// NodeFactory/Datatype/DatatypeNodeFactory
{attribute 'linkalways'} 
{attribute 'no_explicit_call' := 'This FB is a CLASS and must be accessed using methods or properties'}
{attribute 'enable_dynamic_creation'}
FUNCTION_BLOCK DatatypeNodeFactory IMPLEMENTS I_EventHandler
VAR
	datatypes : I_Datatypes;
	nodeFactory : I_NodeFactory;
	selfCreatedNodes : Stack;
END_VAR

METHOD FB_init : BOOL
VAR_INPUT
	bInitRetains : BOOL; // if TRUE, the retain variables are initialized (warm start / cold start)
	bInCopyCode : BOOL;  // if TRUE, the instance afterwards gets moved into the copy code (online change)
	Datatypes : I_Datatypes;
	NodeFactory : I_NodeFactory;	
END_VAR
THIS^.datatypes := Datatypes;
THIS^.nodeFactory := NodeFactory;

RegisterWithDatatypes();
END_METHOD

METHOD FB_exit : BOOL
VAR_INPUT
	bInCopyCode : BOOL; // if TRUE, the exit method is called for exiting an instance that is copied afterwards (online change).
END_VAR
IF bInCopyCode THEN
	RETURN;
END_IF

DeregisterWithDatatypes();
DisposeSelfCreatedNodes();
END_METHOD

METHOD PRIVATE DeregisterWithDatatypes
VAR_INPUT
END_VAR
IF datatypes = 0 THEN
	RETURN;
END_IF

datatypes.OffEvent('OnDatatypeAdded', THIS^);
datatypes := 0;
END_METHOD

METHOD PRIVATE DisposeSelfCreatedNodes : BOOL
VAR
	node : I_Node;
END_VAR
WHILE selfCreatedNodes.TryPop(node) DO
	node.Dispose();
END_WHILE
END_METHOD

METHOD PRIVATE RegisterWithDatatypes
VAR_INPUT
END_VAR
IF datatypes = 0 THEN
	RETURN;
END_IF

datatypes.OnEvent('OnDatatypeAdded', THIS^);
END_METHOD

METHOD PROTECTED CreateAliasArrayBundleNode : I_Node
VAR_INPUT
	NodeDatatype : I_AliasDatatype;
END_VAR
VAR
	pAnyBundleNode : POINTER TO AnyAliasArrayBundleNode;
END_VAR
pAnyBundleNode := __NEW(AnyAliasArrayBundleNode(AliasDatatype := NodeDatatype));
CreateAliasArrayBundleNode := pAnyBundleNode^;
END_METHOD

METHOD PROTECTED CreateAliasArrayUnbundleNode : I_Node
VAR_INPUT
	NodeDatatype : I_AliasDatatype;
END_VAR
VAR
	pAnyUnbundleNode : POINTER TO AnyAliasArrayUnbundleNode;
END_VAR
pAnyUnbundleNode := __NEW(AnyAliasArrayUnbundleNode(AliasDatatype := NodeDatatype));
CreateAliasArrayUnbundleNode := pAnyUnbundleNode^;
END_METHOD

METHOD PROTECTED CreateAliasStructureBundleNode : I_Node
VAR_INPUT
	NodeDatatype : I_AliasDatatype;
END_VAR
VAR
	pAnyBundleNode : POINTER TO AnyAliasStructureBundleNode;
END_VAR
pAnyBundleNode := __NEW(AnyAliasStructureBundleNode(AliasDatatype := NodeDatatype));
CreateAliasStructureBundleNode := pAnyBundleNode^;
END_METHOD

METHOD PROTECTED CreateAliasStructureUnbundleNode : I_Node
VAR_INPUT
	NodeDatatype : I_AliasDatatype;
END_VAR
VAR
	pAnyUnbundleNode : POINTER TO AnyAliasStructureUnbundleNode;
END_VAR
pAnyUnbundleNode := __NEW(AnyAliasStructureUnbundleNode(AliasDatatype := NodeDatatype));
CreateAliasStructureUnbundleNode := pAnyUnbundleNode^;
END_METHOD

METHOD PROTECTED CreateArrayBundleNode : I_Node
VAR_INPUT
	NodeDatatype : I_ArrayDatatype;
END_VAR
VAR
	pAnyBundleNode : POINTER TO AnyArrayBundleNode;
END_VAR
pAnyBundleNode := __NEW(AnyArrayBundleNode(ArrayDatatype := NodeDatatype));
CreateArrayBundleNode := pAnyBundleNode^;
END_METHOD

METHOD PROTECTED CreateArrayUnbundleNode : I_Node
VAR_INPUT
	NodeDatatype : I_ArrayDatatype;
END_VAR
VAR
	pAnyUnbundleNode : POINTER TO AnyArrayUnbundleNode;
END_VAR
pAnyUnbundleNode := __NEW(AnyArrayUnbundleNode(ArrayDatatype := NodeDatatype));
CreateArrayUnbundleNode := pAnyUnbundleNode^;
END_METHOD

METHOD PROTECTED CreateDisplayNode : I_Node
VAR_INPUT
	NodeDatatype : I_Datatype;
END_VAR
VAR
	pAnyDisplayNode : POINTER TO AnyDisplayNode;
END_VAR
pAnyDisplayNode := __NEW(AnyDisplayNode(Datatype := NodeDatatype));
CreateDisplayNode := pAnyDisplayNode^;
END_METHOD

METHOD PROTECTED CreateInterfaceDisplayNode : I_Node
VAR_INPUT
	NodeDatatype : I_InterfaceDatatype;
END_VAR
VAR
	pAnyInterfaceDisplayNode : POINTER TO AnyInterfaceDisplayNode;
END_VAR
pAnyInterfaceDisplayNode := __NEW(AnyInterfaceDisplayNode(Datatype := NodeDatatype));
CreateInterfaceDisplayNode := pAnyInterfaceDisplayNode^;
END_METHOD

METHOD PROTECTED CreateLiteralNode : I_Node
VAR_INPUT
	NodeDatatype : I_Datatype;
END_VAR
VAR
	pAnyLiteralNode : POINTER TO AnyLiteralNode;
END_VAR
pAnyLiteralNode := __NEW(AnyLiteralNode(Datatype := NodeDatatype));
CreateLiteralNode := pAnyLiteralNode^;
END_METHOD

METHOD PROTECTED CreateStructureBundleNode : I_Node
VAR_INPUT
	NodeDatatype : I_StructuredDatatype;
END_VAR
VAR
	pAnyBundleNode : POINTER TO AnyStructureBundleNode;
END_VAR
pAnyBundleNode := __NEW(AnyStructureBundleNode(StructuredDatatype := NodeDatatype));
CreateStructureBundleNode := pAnyBundleNode^;
END_METHOD

METHOD PROTECTED CreateStructureUnbundleNode : I_Node
VAR_INPUT
	NodeDatatype : I_StructuredDatatype;
END_VAR
VAR
	pAnyUnbundleNode : POINTER TO AnyStructureUnbundleNode;
END_VAR
pAnyUnbundleNode := __NEW(AnyStructureUnbundleNode(StructuredDatatype := NodeDatatype));
CreateStructureUnbundleNode := pAnyUnbundleNode^;
END_METHOD

METHOD PROTECTED RegisterAliasArrayBundleNodeOfType
VAR_INPUT
	AliasDatatype : I_AliasDatatype;
END_VAR
VAR
	node : I_Node;
	path : T_MAXSTRING;
END_VAR
node := CreateAliasArrayBundleNode(AliasDatatype);
selfCreatedNodes.Push(node);
path := concat('Bundle/', AliasDatatype.Identifier);
nodeFactory.AddNodeAsPrototype(path,node);
END_METHOD

METHOD PROTECTED RegisterAliasArrayUnbundleNodeOfType
VAR_INPUT
	AliasDatatype : I_AliasDatatype;
END_VAR
VAR
	node : I_Node;
	path : T_MAXSTRING;
END_VAR
node := CreateAliasArrayUnbundleNode(AliasDatatype);
selfCreatedNodes.Push(node);
path := concat('Unbundle/', AliasDatatype.Identifier);
nodeFactory.AddNodeAsPrototype(path,node);
END_METHOD

METHOD PROTECTED RegisterAliasStructureBundleNodeOfType
VAR_INPUT
	AliasDatatype : I_AliasDatatype;
END_VAR
VAR
	node : I_Node;
	path : T_MAXSTRING;
END_VAR
node := CreateAliasStructureBundleNode(AliasDatatype);
selfCreatedNodes.Push(node);
path := concat('Bundle/', AliasDatatype.Identifier);
nodeFactory.AddNodeAsPrototype(path,node);
END_METHOD

METHOD PROTECTED RegisterAliasStructureUnbundleNodeOfType
VAR_INPUT
	AliasDatatype : I_AliasDatatype;
END_VAR
VAR
	node : I_Node;
	path : T_MAXSTRING;
END_VAR
node := CreateAliasStructureUnbundleNode(AliasDatatype);
selfCreatedNodes.Push(node);
path := concat('Unbundle/', AliasDatatype.Identifier);
nodeFactory.AddNodeAsPrototype(path,node);
END_METHOD

METHOD PROTECTED RegisterArrayBundleNodeOfType
VAR_INPUT
	NodeDatatype : I_ArrayDatatype;
END_VAR
VAR
	node : I_Node;
	path : T_MAXSTRING;
END_VAR
node := CreateArrayBundleNode(NodeDatatype);
selfCreatedNodes.Push(node);
path := concat('Bundle/', NodeDatatype.Identifier);
nodeFactory.AddNodeAsPrototype(path,node);
END_METHOD

METHOD PROTECTED RegisterArrayUnbundleNodeOfType
VAR_INPUT
	NodeDatatype : I_ArrayDatatype;
END_VAR
VAR
	node : I_Node;
	path : T_MAXSTRING;
END_VAR
node := CreateArrayUnbundleNode(NodeDatatype);
selfCreatedNodes.Push(node);
path := concat('Unbundle/', NodeDatatype.Identifier);
nodeFactory.AddNodeAsPrototype(path,node);
END_METHOD

METHOD PROTECTED RegisterInterfaceDisplayNodeOfType
VAR_INPUT
	NodeDatatype : I_InterfaceDatatype;
END_VAR
VAR
	node : I_Node;
	path : T_MAXSTRING;
END_VAR
node := CreateInterfaceDisplayNode(NodeDatatype);
selfCreatedNodes.Push(node);
path := concat('Display/', NodeDatatype.Identifier);
nodeFactory.AddNodeAsPrototype(path,node);
END_METHOD

METHOD PROTECTED RegisterInterfaceLiteralNodeOfType
VAR_INPUT
	NodeDatatype : I_InterfaceDatatype;
END_VAR
VAR
	node : I_Node;
	path : T_MAXSTRING;
END_VAR
node := CreateLiteralNode(NodeDatatype);
selfCreatedNodes.Push(node);
path := concat('Literal/', NodeDatatype.Identifier);
nodeFactory.AddNodeAsPrototype(path,node);
END_METHOD

METHOD PROTECTED RegisterPrimitiveDisplayNodeOfType
VAR_INPUT
	NodeDatatype : I_Datatype;
END_VAR
VAR
	node : I_Node;
	path : T_MAXSTRING;
END_VAR
node := CreateDisplayNode(NodeDatatype);
selfCreatedNodes.Push(node);
path := concat('Display/', NodeDatatype.TypeName);
nodeFactory.AddNodeAsPrototype(path,node);
END_METHOD

METHOD PROTECTED RegisterPrimitiveLiteralNodeOfType
VAR_INPUT
	NodeDatatype : I_Datatype;
END_VAR
VAR
	node : I_Node;
	path : T_MAXSTRING;
END_VAR
node := CreateLiteralNode(NodeDatatype);
selfCreatedNodes.Push(node);
path := concat('Literal/', NodeDatatype.TypeName);
nodeFactory.AddNodeAsPrototype(path,node);
END_METHOD

METHOD PROTECTED RegisterStructureBundleNodeOfType
VAR_INPUT
	NodeDatatype : I_StructuredDatatype;
END_VAR
VAR
	node : I_Node;
	path : T_MAXSTRING;
END_VAR
node := CreateStructureBundleNode(NodeDatatype);
selfCreatedNodes.Push(node);
path := concat('Bundle/', NodeDatatype.Identifier);
nodeFactory.AddNodeAsPrototype(path,node);
END_METHOD

METHOD PROTECTED RegisterStructureUnbundleNodeOfType
VAR_INPUT
	NodeDatatype : I_StructuredDatatype;
END_VAR
VAR
	node : I_Node;
	path : T_MAXSTRING;
END_VAR
node := CreateStructureUnbundleNode(NodeDatatype);
selfCreatedNodes.Push(node);
path := concat('Unbundle/', NodeDatatype.Identifier);
nodeFactory.AddNodeAsPrototype(path,node);
END_METHOD

METHOD PROTECTED RegisterUdtDisplayNodeOfType
VAR_INPUT
	NodeDatatype : I_UserDefinedDatatype;
END_VAR
VAR
	node : I_Node;
	path : T_MAXSTRING;
END_VAR
node := CreateDisplayNode(NodeDatatype);
selfCreatedNodes.Push(node);
path := concat('Display/', NodeDatatype.Identifier);
nodeFactory.AddNodeAsPrototype(path,node);
END_METHOD

METHOD PROTECTED RegisterUdtLiteralNodeOfType
VAR_INPUT
	NodeDatatype : I_UserDefinedDatatype;
END_VAR
VAR
	node : I_Node;
	path : T_MAXSTRING;
END_VAR
node := CreateLiteralNode(NodeDatatype);
selfCreatedNodes.Push(node);
path := concat('Literal/', NodeDatatype.Identifier);
nodeFactory.AddNodeAsPrototype(path,node);
END_METHOD

METHOD PUBLIC HandleEvent
VAR_INPUT
	Event : I_Event;
END_VAR
VAR
	datatypeAddedEvent : I_DatatypeAddedEvent;
	primitiveDatatype : I_Datatype;
	aliasDatatypeAddedEvent : I_AliasDatatypeAddedEvent;
	aliasDatatype : I_AliasDatatype;
	enumDatatypeAddedEvent : I_EnumDatatypeAddedEvent;
	enumDatatype : I_EnumDatatype;
	structuredDatatypeAddedEvent : I_StructuredDatatypeAddedEvent;
	structureDatatype : I_StructuredDatatype;
	interfaceDatatypeAddedEvent : I_InterfaceDatatypeAddedEvent;
	interfaceDatatype : I_InterfaceDatatype;
	arrayDatatypeAddedEvent : I_ArrayDatatypeAddedEvent;
	arrayDatatype : I_ArrayDatatype;
END_VAR
IF __QUERYINTERFACE(event, aliasDatatypeAddedEvent) THEN
	aliasDatatype := aliasDatatypeAddedEvent.Target;
	RegisterUdtLiteralNodeOfType(aliasDatatype);
	RegisterUdtDisplayNodeOfType(aliasDatatype);
	
	// at this point we have the lowest level alias who's base type is not alias (or we reached a breakout)
	IF aliasDatatype.Root.TryResolveAsArrayDatatype(arrayDatatype) THEN
		RegisterAliasArrayBundleNodeOfType(aliasDatatype);
		RegisterAliasArrayUnbundleNodeOfType(aliasDatatype);
	ELSIF aliasDatatype.Root.TryResolveAsStructuredDatatype(structureDatatype) THEN
		RegisterAliasStructureBundleNodeOfType(aliasDatatype);
		RegisterAliasStructureUnbundleNodeOfType(aliasDatatype);
	END_IF
		
	RETURN;
END_IF

IF __QUERYINTERFACE(event, enumDatatypeAddedEvent) THEN
	enumDatatype := enumDatatypeAddedEvent.Target;
	RegisterUdtLiteralNodeOfType(enumDatatype);
	RegisterUdtDisplayNodeOfType(enumDatatype);
	RETURN;
END_IF

IF __QUERYINTERFACE(event, interfaceDatatypeAddedEvent) THEN
	interfaceDatatype := interfaceDatatypeAddedEvent.Target;
	RegisterInterfaceLiteralNodeOfType(interfaceDatatype);
	RegisterInterfaceDisplayNodeOfType(interfaceDatatype);
	RETURN;
END_IF

IF __QUERYINTERFACE(event, structuredDatatypeAddedEvent) THEN
	structureDatatype := structuredDatatypeAddedEvent.Target;
	RegisterUdtLiteralNodeOfType(structureDatatype);
	RegisterUdtDisplayNodeOfType(structureDatatype);
	RegisterStructureBundleNodeOfType(structureDatatype);
	RegisterStructureUnbundleNodeOfType(structureDatatype);
	RETURN;
END_IF

IF __QUERYINTERFACE(event, arrayDatatypeAddedEvent) THEN
	RegisterUdtLiteralNodeOfType(arrayDatatypeAddedEvent.Target);
	RegisterUdtDisplayNodeOfType(arrayDatatypeAddedEvent.Target);
	RegisterArrayBundleNodeOfType(arrayDatatypeAddedEvent.Target);
	RegisterArrayUnbundleNodeOfType(arrayDatatypeAddedEvent.Target);
	RETURN;
END_IF

IF __QUERYINTERFACE(event, datatypeAddedEvent) THEN
	primitiveDatatype := datatypeAddedEvent.Target;
	RegisterPrimitiveLiteralNodeOfType(primitiveDatatype);
	RegisterPrimitiveDisplayNodeOfType(primitiveDatatype);
	RETURN;
END_IF
END_METHOD

END_FUNCTION_BLOCK

// Node/Bundle/AnyAliasArrayBundleNode
{attribute 'linkalways'} 
{attribute 'no_explicit_call' := 'This FB is a CLASS and must be accessed using methods or properties'}
{attribute 'enable_dynamic_creation'}
FUNCTION_BLOCK FINAL AnyAliasArrayBundleNode EXTENDS Node
VAR
	in : I_AliasDatatype;
	out : I_AliasDatatype;
	datatypeOperations : DatatypeOperations;
	selfMadeElements : Stack;
END_VAR

METHOD FB_init : BOOL
VAR_INPUT
	bInitRetains : BOOL; // if TRUE, the retain variables are initialized (warm start / cold start)
	bInCopyCode : BOOL;  // if TRUE, the instance afterwards gets moved into the copy code (online change)
	AliasDatatype : I_AliasDatatype;
END_VAR
VAR
	inAsArray : I_ArrayDatatype;
	inAs1D : I_ArrayDatatype_1D;
	inAs2D : I_ArrayDatatype_2D;
	inAs3D : I_ArrayDatatype_3D;
END_VAR
AliasDatatype.Clone().TryResolveAsAliasDatatype(out);
AddOutput('out', out);

AliasDatatype.Clone().TryResolveAsAliasDatatype(in);
in.Root.TryResolveAsArrayDatatype(inAsArray);

IF inAsArray.TryResolveAs1DArrayDatatype(inAs1D) THEN
	ConfigureFor1DArray(inAs1D);
ELSIF inAsArray.TryResolveAs2DArrayDatatype(inAs2D) THEN
	ConfigureFor2DArray(inAs2D);
ELSIF inAsArray.TryResolveAs3DArrayDatatype(inAs3D) THEN
	ConfigureFor3DArray(inAs3D);
END_IF
END_METHOD

METHOD FB_exit : BOOL
VAR_INPUT
	bInCopyCode : BOOL; // if TRUE, the exit method is called for exiting an instance that is copied afterwards (online change).
END_VAR
VAR
	element : I_Datatype;
END_VAR
IF bInCopyCode THEN
	RETURN;
END_IF

in.Dispose();
out.Dispose();
datatypeOperations.Clear();

WHILE selfMadeElements.TryPop(element) DO
	IF element <> 0 THEN 
		element.Dispose();
	END_IF
END_WHILE
END_METHOD

METHOD PRIVATE ConfigureFor1DArray
VAR_INPUT
	array1D : I_ArrayDatatype_1D;
END_VAR
VAR
	lowerBound : DINT;
	upperBound : DINT;
	i : DINT;
	element : I_Datatype;
	elementClone : I_Datatype;
END_VAR
IF NOT array1D.TryGetLowerBound(1, lowerBound) THEN
	RETURN;
END_IF

IF NOT array1D.TryGetUpperBound(1, upperBound) THEN
	RETURN;
END_IF

FOR i := lowerBound TO upperBound DO
	
	IF array1D.TryGetElementAsDatatypeByIndex(i, element) THEN
		elementClone := element.Clone();
		datatypeOperations.AddMemoryCopyOperation(elementClone, element);
		AddParameter(Get1DIndexName(i), elementClone);
		selfMadeElements.Push(elementClone);
	END_IF
	
END_FOR
END_METHOD

METHOD PRIVATE ConfigureFor2DArray
VAR_INPUT
	array2D : I_ArrayDatatype_2D;
END_VAR
VAR
	lowerBoundD1 : DINT;
	upperBoundD1 : DINT;
	lowerBoundD2 : DINT;
	upperBoundD2 : DINT;
	i, j : DINT;
	element : I_Datatype;
	elementClone : I_Datatype;
END_VAR
IF NOT array2D.TryGetLowerBound(1, lowerBoundD1) THEN
	RETURN;
END_IF

IF NOT array2D.TryGetUpperBound(1, upperBoundD1) THEN
	RETURN;
END_IF

IF NOT array2D.TryGetLowerBound(2, lowerBoundD2) THEN
	RETURN;
END_IF

IF NOT array2D.TryGetUpperBound(2, upperBoundD2) THEN
	RETURN;
END_IF

FOR i := lowerBoundD1 TO upperBoundD1 DO
	FOR j := lowerBoundD2 TO upperBoundD2 DO
	
		IF array2D.TryGetElementAsDatatypeByIndex(i, j, element) THEN
			elementClone := element.Clone();
			datatypeOperations.AddMemoryCopyOperation(elementClone, element);
			AddParameter(Get2DIndexName(i,j), elementClone);
			selfMadeElements.Push(elementClone);
		END_IF
	
	END_FOR
END_FOR
END_METHOD

METHOD PRIVATE ConfigureFor3DArray
VAR_INPUT
	array3D : I_ArrayDatatype_3D;
END_VAR
VAR
	lowerBoundD1 : DINT;
	upperBoundD1 : DINT;
	lowerBoundD2 : DINT;
	upperBoundD2 : DINT;
	lowerBoundD3 : DINT;
	upperBoundD3 : DINT;
	i, j, k : DINT;
	element : I_Datatype;
	elementClone : I_Datatype;
END_VAR
IF NOT array3D.TryGetLowerBound(1, lowerBoundD1) THEN
	RETURN;
END_IF

IF NOT array3D.TryGetUpperBound(1, upperBoundD1) THEN
	RETURN;
END_IF

IF NOT array3D.TryGetLowerBound(2, lowerBoundD2) THEN
	RETURN;
END_IF

IF NOT array3D.TryGetUpperBound(2, upperBoundD2) THEN
	RETURN;
END_IF

IF NOT array3D.TryGetLowerBound(3, lowerBoundD3) THEN
	RETURN;
END_IF

IF NOT array3D.TryGetUpperBound(3, upperBoundD3) THEN
	RETURN;
END_IF

FOR i := lowerBoundD1 TO upperBoundD1 DO
	FOR j := lowerBoundD2 TO upperBoundD2 DO
		FOR k := lowerBoundD3 TO upperBoundD3 DO
	
			IF array3D.TryGetElementAsDatatypeByIndex(i, j, k, element) THEN
				elementClone := element.Clone();
				datatypeOperations.AddMemoryCopyOperation(elementClone, element);
				AddParameter(Get3DIndexName(i, j, k), elementClone);
				selfMadeElements.Push(elementClone);
			END_IF
			
		END_FOR
	END_FOR
END_FOR
END_METHOD

METHOD PRIVATE Get1DIndexName : T_MAXSTRING
VAR_INPUT
	Index : DINT;
END_VAR
Get1DIndexName := concat('[', DINT_TO_STRING(Index));
Get1DIndexName := concat(Get1DIndexName, ']');
END_METHOD

METHOD PRIVATE Get2DIndexName : T_MAXSTRING
VAR_INPUT
	Index1 : DINT;
	Index2 : DINT;
END_VAR
Get2DIndexName := concat('[', DINT_TO_STRING(Index1));
Get2DIndexName := concat(Get2DIndexName, ',');
Get2DIndexName := concat(Get2DIndexName, DINT_TO_STRING(Index2));
Get2DIndexName := concat(Get2DIndexName, ']');
END_METHOD

METHOD PRIVATE Get3DIndexName : T_MAXSTRING
VAR_INPUT
	Index1 : DINT;
	Index2 : DINT;
	Index3 : DINT;
END_VAR
Get3DIndexName := concat('[',DINT_TO_STRING(Index1));
Get3DIndexName := concat(Get3DIndexName,',');
Get3DIndexName := concat(Get3DIndexName,DINT_TO_STRING(Index2));
Get3DIndexName := concat(Get3DIndexName,',');
Get3DIndexName := concat(Get3DIndexName,DINT_TO_STRING(Index3));
Get3DIndexName := concat(Get3DIndexName,']');
END_METHOD

METHOD PUBLIC Clone : I_Node
VAR
	pNode : POINTER TO AnyAliasArrayBundleNode;
END_VAR
pNode := __NEW(AnyAliasArrayBundleNode(AliasDatatype := in));
Clone := pNode^;
END_METHOD

METHOD PROTECTED OnExecute
VAR
END_VAR
datatypeOperations.Execute();
memcpy(out.Address, in.Address, in.Size);
END_METHOD

END_FUNCTION_BLOCK

// Node/Unbundle/AnyAliasArrayUnbundleNode
{attribute 'linkalways'} 
{attribute 'no_explicit_call' := 'This FB is a CLASS and must be accessed using methods or properties'}
{attribute 'enable_dynamic_creation'}
FUNCTION_BLOCK FINAL AnyAliasArrayUnbundleNode EXTENDS Node
VAR
	in : I_AliasDatatype;
	out : I_AliasDatatype;
	datatypeOperations : DatatypeOperations;
	selfMadeElements : Stack;
END_VAR

METHOD FB_init : BOOL
VAR_INPUT
	bInitRetains : BOOL; // if TRUE, the retain variables are initialized (warm start / cold start)
	bInCopyCode : BOOL;  // if TRUE, the instance afterwards gets moved into the copy code (online change)
	AliasDatatype : I_AliasDatatype;
END_VAR
VAR
	outAsArray : I_ArrayDatatype;
	outAs1D : I_ArrayDatatype_1D;
	outAs2D : I_ArrayDatatype_2D;
	outAs3D : I_ArrayDatatype_3D;
END_VAR
AliasDatatype.Clone().TryResolveAsAliasDatatype(in);
AddInput('in', in);

AliasDatatype.Clone().TryResolveAsAliasDatatype(out);
out.Root.TryResolveAsArrayDatatype(outAsArray);

IF outAsArray.TryResolveAs1DArrayDatatype(outAs1D) THEN
	ConfigureFor1DArray(outAs1D);
ELSIF outAsArray.TryResolveAs2DArrayDatatype(outAs2D) THEN
	ConfigureFor2DArray(outAs2D);
ELSIF outAsArray.TryResolveAs3DArrayDatatype(outAs3D) THEN
	ConfigureFor3DArray(outAs3D);
END_IF
END_METHOD

METHOD FB_exit : BOOL
VAR_INPUT
	bInCopyCode : BOOL; // if TRUE, the exit method is called for exiting an instance that is copied afterwards (online change).
END_VAR
VAR
	element : I_Datatype;
END_VAR
IF bInCopyCode THEN
	RETURN;
END_IF

in.Dispose();
out.Dispose();
datatypeOperations.Clear();

WHILE selfMadeElements.TryPop(element) DO
	IF element <> 0 THEN 
		element.dispose();
	END_IF
END_WHILE
END_METHOD

METHOD PRIVATE ConfigureFor1DArray
VAR_INPUT
	array1D : I_ArrayDatatype_1D;
END_VAR
VAR
	lowerBound : DINT;
	upperBound : DINT;
	i : DINT;
	element : I_Datatype;
	elementClone : I_Datatype;
END_VAR
IF NOT array1D.TryGetLowerBound(1, lowerBound) THEN
	RETURN;
END_IF

IF NOT array1D.TryGetUpperBound(1, upperBound) THEN
	RETURN;
END_IF

FOR i := lowerBound TO upperBound DO
	
	IF array1D.TryGetElementAsDatatypeByIndex(i, element) THEN
		elementClone := element.Clone();
		datatypeOperations.AddMemoryCopyOperation(element, elementClone);
		AddOutput(Get1DIndexName(i), elementClone);
		selfMadeElements.Push(elementClone);
	END_IF
	
END_FOR
END_METHOD

METHOD PRIVATE ConfigureFor2DArray
VAR_INPUT
	array2D : I_ArrayDatatype_2D;
END_VAR
VAR
	lowerBoundD1 : DINT;
	upperBoundD1 : DINT;
	lowerBoundD2 : DINT;
	upperBoundD2 : DINT;
	i, j : DINT;
	element : I_Datatype;
	elementClone : I_Datatype;
END_VAR
IF NOT array2D.TryGetLowerBound(1, lowerBoundD1) THEN
	RETURN;
END_IF

IF NOT array2D.TryGetUpperBound(1, upperBoundD1) THEN
	RETURN;
END_IF

IF NOT array2D.TryGetLowerBound(2, lowerBoundD2) THEN
	RETURN;
END_IF

IF NOT array2D.TryGetUpperBound(2, upperBoundD2) THEN
	RETURN;
END_IF

FOR i := lowerBoundD1 TO upperBoundD1 DO
	FOR j := lowerBoundD2 TO upperBoundD2 DO
	
		IF array2D.TryGetElementAsDatatypeByIndex(i, j, element) THEN
			elementClone := element.Clone();
			datatypeOperations.AddMemoryCopyOperation(element, elementClone);
			AddOutput(Get2DIndexName(i,j), elementClone);
			selfMadeElements.Push(elementClone);
		END_IF
	
	END_FOR
END_FOR
END_METHOD

METHOD PRIVATE ConfigureFor3DArray
VAR_INPUT
	array3D : I_ArrayDatatype_3D;
END_VAR
VAR
	lowerBoundD1 : DINT;
	upperBoundD1 : DINT;
	lowerBoundD2 : DINT;
	upperBoundD2 : DINT;
	lowerBoundD3 : DINT;
	upperBoundD3 : DINT;
	i, j, k : DINT;
	element : I_Datatype;
	elementClone : I_Datatype;
END_VAR
IF NOT array3D.TryGetLowerBound(1, lowerBoundD1) THEN
	RETURN;
END_IF

IF NOT array3D.TryGetUpperBound(1, upperBoundD1) THEN
	RETURN;
END_IF

IF NOT array3D.TryGetLowerBound(2, lowerBoundD2) THEN
	RETURN;
END_IF

IF NOT array3D.TryGetUpperBound(2, upperBoundD2) THEN
	RETURN;
END_IF

IF NOT array3D.TryGetLowerBound(3, lowerBoundD3) THEN
	RETURN;
END_IF

IF NOT array3D.TryGetUpperBound(3, upperBoundD3) THEN
	RETURN;
END_IF

FOR i := lowerBoundD1 TO upperBoundD1 DO
	FOR j := lowerBoundD2 TO upperBoundD2 DO
		FOR k := lowerBoundD3 TO upperBoundD3 DO
	
			IF array3D.TryGetElementAsDatatypeByIndex(i, j, k, element) THEN
				elementClone := element.Clone();
				datatypeOperations.AddMemoryCopyOperation(element, elementClone);
				AddOutput(Get3DIndexName(i,j,k), elementClone);
				selfMadeElements.Push(elementClone);
			END_IF
			
		END_FOR
	END_FOR
END_FOR
END_METHOD

METHOD PRIVATE Get1DIndexName : T_MAXSTRING
VAR_INPUT
	Index : DINT;
END_VAR
Get1DIndexName := concat('[',DINT_TO_STRING(Index));
Get1DIndexName := concat(Get1DIndexName,']');
END_METHOD

METHOD PRIVATE Get2DIndexName : T_MAXSTRING
VAR_INPUT
	Index1 : DINT;
	Index2 : DINT;
END_VAR
Get2DIndexName := concat('[',DINT_TO_STRING(Index1));
Get2DIndexName := concat(Get2DIndexName,',');
Get2DIndexName := concat(Get2DIndexName,DINT_TO_STRING(Index2));
Get2DIndexName := concat(Get2DIndexName,']');
END_METHOD

METHOD PRIVATE Get3DIndexName : T_MAXSTRING
VAR_INPUT
	Index1 : DINT;
	Index2 : DINT;
	Index3 : DINT;
END_VAR
Get3DIndexName := concat('[',DINT_TO_STRING(Index1));
Get3DIndexName := concat(Get3DIndexName,',');
Get3DIndexName := concat(Get3DIndexName,DINT_TO_STRING(Index2));
Get3DIndexName := concat(Get3DIndexName,',');
Get3DIndexName := concat(Get3DIndexName,DINT_TO_STRING(Index3));
Get3DIndexName := concat(Get3DIndexName,']');
END_METHOD

METHOD PUBLIC Clone : I_Node
VAR
	pNode : POINTER TO AnyAliasArrayUnbundleNode;
END_VAR
pNode := __NEW(AnyAliasArrayUnbundleNode(AliasDatatype := in));
Clone := pNode^;
END_METHOD

METHOD PROTECTED OnExecute
VAR
END_VAR
memcpy(out.Address, in.Address, in.Size);
datatypeOperations.Execute();
END_METHOD

END_FUNCTION_BLOCK

// Node/Bundle/AnyAliasStructureBundleNode
{attribute 'linkalways'} 
{attribute 'no_explicit_call' := 'This FB is a CLASS and must be accessed using methods or properties'}
{attribute 'enable_dynamic_creation'}
FUNCTION_BLOCK FINAL AnyAliasStructureBundleNode EXTENDS Node
VAR
	in : I_AliasDatatype;
	out : I_AliasDatatype;
	datatypeOperations : DatatypeOperations;
	selfMadeMembers : Stack;
END_VAR

METHOD FB_init : BOOL
VAR_INPUT
	bInitRetains : BOOL; // if TRUE, the retain variables are initialized (warm start / cold start)
	bInCopyCode : BOOL;  // if TRUE, the instance afterwards gets moved into the copy code (online change)
	AliasDatatype : I_AliasDatatype;
END_VAR
VAR
	inAsStructured : I_StructuredDatatype;
	enumerator : I_KeyValueForwardEnumerator;
	member : I_Datatype;
	memberAsBit : I_BIT;
	memberAsBool : I_Datatype;
	_bool : pointer to _BOOL;
	memberClone : I_Datatype;
END_VAR
AliasDatatype.Clone().TryResolveAsAliasDatatype(out);
AddOutput('out', out);

AliasDatatype.Clone().TryResolveAsAliasDatatype(in);
in.Root.TryResolveAsStructuredDatatype(inAsStructured);
enumerator := inAsStructured.Members.GetMemberEnumerator();

WHILE enumerator.MoveNext() DO 
	IF enumerator.TryGet(member) THEN
		IF member.TryResolveAs_BIT(memberAsBit) THEN
			// if the element is a _bit then this needs to be treated differently (as you cannot simply memcpy
			// a bit, as it sits next to other data. Instead, a bool is added in it's place.	
			_bool := __NEW(_BOOL(InitialValue := memberAsBit.Value));
			datatypeOperations.AddWriteBoolToBitOperation(_bool^, memberAsBit);
			AddParameter(enumerator.Key, _bool^);
			memberAsBool := _bool^;
			selfMadeMembers.Push(memberAsBool);
		ELSE
			// for all other datatypes,
			memberClone := member.Clone();
			datatypeOperations.AddMemoryCopyOperation(memberClone, member);
			AddParameter(enumerator.key, memberClone);
			selfMadeMembers.Push(memberClone);
		END_IF
	END_IF
END_WHILE

enumerator.Dispose();
END_METHOD

METHOD FB_exit : BOOL
VAR_INPUT
	bInCopyCode : BOOL; // if TRUE, the exit method is called for exiting an instance that is copied afterwards (online change).
END_VAR
VAR
	member : I_Datatype;
END_VAR
IF bInCopyCode THEN
	RETURN;
END_IF

in.Dispose();
out.Dispose();
datatypeOperations.Clear();

WHILE selfMadeMembers.TryPop(member) DO
	IF member <> 0 THEN 
		member.dispose();
	END_IF
END_WHILE
END_METHOD

METHOD PUBLIC Clone : I_Node
VAR
	pNode : POINTER TO AnyAliasStructureBundleNode;
END_VAR
pNode := __NEW(AnyAliasStructureBundleNode(AliasDatatype := in));
Clone := pNode^;
END_METHOD

METHOD PROTECTED OnExecute
VAR
END_VAR
datatypeOperations.Execute();
memcpy(out.Address, in.Address, in.Size);
END_METHOD

END_FUNCTION_BLOCK

// Node/Unbundle/AnyAliasStructureUnbundleNode
{attribute 'linkalways'} 
{attribute 'no_explicit_call' := 'This FB is a CLASS and must be accessed using methods or properties'}
{attribute 'enable_dynamic_creation'}
FUNCTION_BLOCK FINAL AnyAliasStructureUnbundleNode EXTENDS Node
VAR
	in : I_AliasDatatype;
	out : I_AliasDatatype;
	datatypeOperations : DatatypeOperations;
	selfMadeMembers : Stack;
END_VAR

METHOD FB_init : BOOL
VAR_INPUT
	bInitRetains : BOOL; // if TRUE, the retain variables are initialized (warm start / cold start)
	bInCopyCode : BOOL;  // if TRUE, the instance afterwards gets moved into the copy code (online change)
	AliasDatatype : I_AliasDatatype;
END_VAR
VAR
	outAsStructure : I_StructuredDatatype;
	enumerator : I_KeyValueForwardEnumerator;
	member : I_Datatype;
	memberAsBit : I_BIT;
	memberAsBool : I_Datatype;
	_bool : Pointer to _BOOL;
	memberClone : I_Datatype;
END_VAR
AliasDatatype.Clone().TryResolveAsAliasDatatype(in);
AddInput('in', in);

AliasDatatype.Clone().TryResolveAsAliasDatatype(out);
out.Root.TryResolveAsStructuredDatatype(outAsStructure);
enumerator := outAsStructure.Members.GetMemberEnumerator();

WHILE enumerator.MoveNext() DO 
	IF enumerator.TryGet(member) THEN
		IF member.TryResolveAs_BIT(memberAsBit) THEN
			// if the element is a _bit then this needs to be treated differently (as you cannot simply memcpy
			// a bit, as it sits next to other data. Instead, a bool is added in it's place.	
			_bool := __NEW(_BOOL(InitialValue := memberAsBit.Value));
			datatypeOperations.AddWriteBitToBoolOperation(memberAsBit, _bool^);
			AddOutput(enumerator.Key, _bool^);
			memberAsBool := _bool^;
			selfMadeMembers.Push(memberAsBool);
		ELSE
			// for all other datatypes,
			memberClone := member.Clone();
			datatypeOperations.AddMemoryCopyOperation(member, memberClone);
			AddOutput(enumerator.key, memberClone);
			selfMadeMembers.Push(memberClone);
		END_IF		
	END_IF
END_WHILE

enumerator.Dispose();
END_METHOD

METHOD FB_exit : BOOL
VAR_INPUT
	bInCopyCode : BOOL; // if TRUE, the exit method is called for exiting an instance that is copied afterwards (online change).
END_VAR
VAR
	member : I_Datatype;
END_VAR
IF bInCopyCode THEN
	RETURN;
END_IF

in.Dispose();
out.Dispose();
datatypeOperations.Clear();

WHILE selfMadeMembers.TryPop(member) DO
	IF member <> 0 THEN 
		member.dispose();
	END_IF
END_WHILE
END_METHOD

METHOD PUBLIC Clone : I_Node
VAR
	pNode : POINTER TO AnyAliasStructureUnbundleNode;
END_VAR
pNode := __NEW(AnyAliasStructureUnbundleNode(AliasDatatype := in));
Clone := pNode^;
END_METHOD

METHOD PROTECTED OnExecute
VAR
END_VAR
memcpy(out.Address, in.Address, in.Size);
datatypeOperations.Execute();
END_METHOD

END_FUNCTION_BLOCK

// Node/Bundle/AnyArrayBundleNode
{attribute 'linkalways'} 
{attribute 'no_explicit_call' := 'This FB is a CLASS and must be accessed using methods or properties'}
{attribute 'enable_dynamic_creation'}
FUNCTION_BLOCK FINAL AnyArrayBundleNode EXTENDS Node
VAR
	in : I_ArrayDatatype;
	out : I_ArrayDatatype;
	datatypeOperations : DatatypeOperations;
	selfMadeElements : Stack;
END_VAR

METHOD FB_init : BOOL
VAR_INPUT
	bInitRetains : BOOL; // if TRUE, the retain variables are initialized (warm start / cold start)
	bInCopyCode : BOOL;  // if TRUE, the instance afterwards gets moved into the copy code (online change)
	ArrayDatatype : I_ArrayDatatype;
END_VAR
VAR
	inAs1D : I_ArrayDatatype_1D;
	inAs2D : I_ArrayDatatype_2D;
	inAs3D : I_ArrayDatatype_3D;
END_VAR
ArrayDatatype.Clone().TryResolveAsArrayDatatype(out);
AddOutput('out', out);

ArrayDatatype.Clone().TryResolveAsArrayDatatype(in);

IF in.TryResolveAs1DArrayDatatype(inAs1D) THEN
	ConfigureFor1DArray(inAs1D);
ELSIF in.TryResolveAs2DArrayDatatype(inAs2D) THEN
	ConfigureFor2DArray(inAs2D);
ELSIF in.TryResolveAs3DArrayDatatype(inAs3D) THEN
	ConfigureFor3DArray(inAs3D);
END_IF
END_METHOD

METHOD FB_exit : BOOL
VAR_INPUT
	bInCopyCode : BOOL; // if TRUE, the exit method is called for exiting an instance that is copied afterwards (online change).
END_VAR
VAR
	element : I_Datatype;
END_VAR
IF bInCopyCode THEN
	RETURN;
END_IF

in.Dispose();
out.Dispose();
datatypeOperations.Clear();

WHILE selfMadeElements.TryPop(element) DO
	IF element <> 0 THEN 
		element.dispose();
	END_IF
END_WHILE
END_METHOD

METHOD PRIVATE ConfigureFor1DArray
VAR_INPUT
	array1D : I_ArrayDatatype_1D;
END_VAR
VAR
	lowerBound : DINT;
	upperBound : DINT;
	i : DINT;
	element : I_Datatype;
	elementClone : I_Datatype;
END_VAR
IF NOT array1D.TryGetLowerBound(1, lowerBound) THEN
	RETURN;
END_IF

IF NOT array1D.TryGetUpperBound(1, upperBound) THEN
	RETURN;
END_IF

FOR i := lowerBound TO upperBound DO
	
	IF array1D.TryGetElementAsDatatypeByIndex(i, element) THEN
		elementClone := element.Clone();
		datatypeOperations.AddMemoryCopyOperation(elementClone, element);
		AddParameter(Get1DIndexName(i), elementClone);
		selfMadeElements.Push(elementClone);
	END_IF
	
END_FOR
END_METHOD

METHOD PRIVATE ConfigureFor2DArray
VAR_INPUT
	array2D : I_ArrayDatatype_2D;
END_VAR
VAR
	lowerBoundD1 : DINT;
	upperBoundD1 : DINT;
	lowerBoundD2 : DINT;
	upperBoundD2 : DINT;
	i, j : DINT;
	element : I_Datatype;
	elementClone : I_Datatype;
END_VAR
IF NOT array2D.TryGetLowerBound(1, lowerBoundD1) THEN
	RETURN;
END_IF

IF NOT array2D.TryGetUpperBound(1, upperBoundD1) THEN
	RETURN;
END_IF

IF NOT array2D.TryGetLowerBound(2, lowerBoundD2) THEN
	RETURN;
END_IF

IF NOT array2D.TryGetUpperBound(2, upperBoundD2) THEN
	RETURN;
END_IF

FOR i := lowerBoundD1 TO upperBoundD1 DO
	FOR j := lowerBoundD2 TO upperBoundD2 DO
	
		IF array2D.TryGetElementAsDatatypeByIndex(i, j, element) THEN
			elementClone := element.Clone();
			datatypeOperations.AddMemoryCopyOperation(elementClone, element);
			AddParameter(Get2DIndexName(i,j), elementClone);
			selfMadeElements.Push(elementClone);
		END_IF
	
	END_FOR
END_FOR
END_METHOD

METHOD PRIVATE ConfigureFor3DArray
VAR_INPUT
	array3D : I_ArrayDatatype_3D;
END_VAR
VAR
	lowerBoundD1 : DINT;
	upperBoundD1 : DINT;
	lowerBoundD2 : DINT;
	upperBoundD2 : DINT;
	lowerBoundD3 : DINT;
	upperBoundD3 : DINT;
	i, j, k : DINT;
	element : I_Datatype;
	elementClone : I_Datatype;
END_VAR
IF NOT array3D.TryGetLowerBound(1, lowerBoundD1) THEN
	RETURN;
END_IF

IF NOT array3D.TryGetUpperBound(1, upperBoundD1) THEN
	RETURN;
END_IF

IF NOT array3D.TryGetLowerBound(2, lowerBoundD2) THEN
	RETURN;
END_IF

IF NOT array3D.TryGetUpperBound(2, upperBoundD2) THEN
	RETURN;
END_IF

IF NOT array3D.TryGetLowerBound(3, lowerBoundD3) THEN
	RETURN;
END_IF

IF NOT array3D.TryGetUpperBound(3, upperBoundD3) THEN
	RETURN;
END_IF

FOR i := lowerBoundD1 TO upperBoundD1 DO
	FOR j := lowerBoundD2 TO upperBoundD2 DO
		FOR k := lowerBoundD3 TO upperBoundD3 DO
	
			IF array3D.TryGetElementAsDatatypeByIndex(i, j, k, element) THEN
				elementClone := element.Clone();
				datatypeOperations.AddMemoryCopyOperation(elementClone, element);
				AddParameter(Get3DIndexName(i,j,k), elementClone);
				selfMadeElements.Push(elementClone);
			END_IF
			
		END_FOR
	END_FOR
END_FOR
END_METHOD

METHOD PRIVATE Get1DIndexName : T_MAXSTRING
VAR_INPUT
	Index : DINT;
END_VAR
Get1DIndexName := concat('[',DINT_TO_STRING(Index));
Get1DIndexName := concat(Get1DIndexName,']');
END_METHOD

METHOD PRIVATE Get2DIndexName : T_MAXSTRING
VAR_INPUT
	Index1 : DINT;
	Index2 : DINT;
END_VAR
Get2DIndexName := concat('[',DINT_TO_STRING(Index1));
Get2DIndexName := concat(Get2DIndexName,',');
Get2DIndexName := concat(Get2DIndexName,DINT_TO_STRING(Index2));
Get2DIndexName := concat(Get2DIndexName,']');
END_METHOD

METHOD PRIVATE Get3DIndexName : T_MAXSTRING
VAR_INPUT
	Index1 : DINT;
	Index2 : DINT;
	Index3 : DINT;
END_VAR
Get3DIndexName := concat('[',DINT_TO_STRING(Index1));
Get3DIndexName := concat(Get3DIndexName,',');
Get3DIndexName := concat(Get3DIndexName,DINT_TO_STRING(Index2));
Get3DIndexName := concat(Get3DIndexName,',');
Get3DIndexName := concat(Get3DIndexName,DINT_TO_STRING(Index3));
Get3DIndexName := concat(Get3DIndexName,']');
END_METHOD

METHOD PUBLIC Clone : I_Node
VAR
	pNode : POINTER TO AnyArrayBundleNode;
END_VAR
pNode := __NEW(AnyArrayBundleNode(ArrayDatatype := in));
Clone := pNode^;
END_METHOD

METHOD PROTECTED OnExecute
VAR
END_VAR
datatypeOperations.Execute();
memcpy(out.Address, in.Address, in.Size);
END_METHOD

END_FUNCTION_BLOCK

// Node/Unbundle/AnyArrayUnbundleNode
{attribute 'linkalways'} 
{attribute 'no_explicit_call' := 'This FB is a CLASS and must be accessed using methods or properties'}
{attribute 'enable_dynamic_creation'}
FUNCTION_BLOCK FINAL AnyArrayUnbundleNode EXTENDS Node
VAR
	in : I_ArrayDatatype;
	out : I_ArrayDatatype;
	datatypeOperations : DatatypeOperations;
	selfMadeElements : Stack;
END_VAR

METHOD FB_init : BOOL
VAR_INPUT
	bInitRetains : BOOL; // if TRUE, the retain variables are initialized (warm start / cold start)
	bInCopyCode : BOOL;  // if TRUE, the instance afterwards gets moved into the copy code (online change)
	ArrayDatatype : I_ArrayDatatype;
END_VAR
VAR
	outAs1D : I_ArrayDatatype_1D;
	outAs2D : I_ArrayDatatype_2D;
	outAs3D : I_ArrayDatatype_3D;
END_VAR
ArrayDatatype.Clone().TryResolveAsArrayDatatype(in);
AddInput('in', in);

ArrayDatatype.Clone().TryResolveAsArrayDatatype(out);

IF out.TryResolveAs1DArrayDatatype(outAs1D) THEN
	ConfigureFor1DArray(outAs1D);
ELSIF out.TryResolveAs2DArrayDatatype(outAs2D) THEN
	ConfigureFor2DArray(outAs2D);
ELSIF out.TryResolveAs3DArrayDatatype(outAs3D) THEN
	ConfigureFor3DArray(outAs3D);
END_IF
END_METHOD

METHOD FB_exit : BOOL
VAR_INPUT
	bInCopyCode : BOOL; // if TRUE, the exit method is called for exiting an instance that is copied afterwards (online change).
END_VAR
VAR
	element : I_Datatype;
END_VAR
IF bInCopyCode THEN
	RETURN;
END_IF

in.Dispose();
out.Dispose();
datatypeOperations.Clear();

WHILE selfMadeElements.TryPop(element) DO
	IF element <> 0 THEN 
		element.dispose();
	END_IF
END_WHILE
END_METHOD

METHOD PRIVATE ConfigureFor1DArray
VAR_INPUT
	array1D : I_ArrayDatatype_1D;
END_VAR
VAR
	lowerBound : DINT;
	upperBound : DINT;
	i : DINT;
	element : I_Datatype;
	elementClone : I_Datatype;
END_VAR
IF NOT array1D.TryGetLowerBound(1, lowerBound) THEN
	RETURN;
END_IF

IF NOT array1D.TryGetUpperBound(1, upperBound) THEN
	RETURN;
END_IF

FOR i := lowerBound TO upperBound DO
	
	IF array1D.TryGetElementAsDatatypeByIndex(i, element) THEN
		elementClone := element.Clone();
		datatypeOperations.AddMemoryCopyOperation(element, elementClone);
		AddOutput(Get1DIndexName(i), elementClone);
		selfMadeElements.Push(elementClone);
	END_IF
	
END_FOR
END_METHOD

METHOD PRIVATE ConfigureFor2DArray
VAR_INPUT
	array2D : I_ArrayDatatype_2D;
END_VAR
VAR
	lowerBoundD1 : DINT;
	upperBoundD1 : DINT;
	lowerBoundD2 : DINT;
	upperBoundD2 : DINT;
	i, j : DINT;
	element : I_Datatype;
	elementClone : I_Datatype;
END_VAR
IF NOT array2D.TryGetLowerBound(1, lowerBoundD1) THEN
	RETURN;
END_IF

IF NOT array2D.TryGetUpperBound(1, upperBoundD1) THEN
	RETURN;
END_IF

IF NOT array2D.TryGetLowerBound(2, lowerBoundD2) THEN
	RETURN;
END_IF

IF NOT array2D.TryGetUpperBound(2, upperBoundD2) THEN
	RETURN;
END_IF

FOR i := lowerBoundD1 TO upperBoundD1 DO
	FOR j := lowerBoundD2 TO upperBoundD2 DO
	
		IF array2D.TryGetElementAsDatatypeByIndex(i, j, element) THEN
			elementClone := element.Clone();
			datatypeOperations.AddMemoryCopyOperation(element, elementClone);
			AddOutput(Get2DIndexName(i,j), elementClone);
			selfMadeElements.Push(elementClone);
		END_IF
	
	END_FOR
END_FOR
END_METHOD

METHOD PRIVATE ConfigureFor3DArray
VAR_INPUT
	array3D : I_ArrayDatatype_3D;
END_VAR
VAR
	lowerBoundD1 : DINT;
	upperBoundD1 : DINT;
	lowerBoundD2 : DINT;
	upperBoundD2 : DINT;
	lowerBoundD3 : DINT;
	upperBoundD3 : DINT;
	i, j, k : DINT;
	element : I_Datatype;
	elementClone : I_Datatype;
END_VAR
IF NOT array3D.TryGetLowerBound(1, lowerBoundD1) THEN
	RETURN;
END_IF

IF NOT array3D.TryGetUpperBound(1, upperBoundD1) THEN
	RETURN;
END_IF

IF NOT array3D.TryGetLowerBound(2, lowerBoundD2) THEN
	RETURN;
END_IF

IF NOT array3D.TryGetUpperBound(2, upperBoundD2) THEN
	RETURN;
END_IF

IF NOT array3D.TryGetLowerBound(3, lowerBoundD3) THEN
	RETURN;
END_IF

IF NOT array3D.TryGetUpperBound(3, upperBoundD3) THEN
	RETURN;
END_IF

FOR i := lowerBoundD1 TO upperBoundD1 DO
	FOR j := lowerBoundD2 TO upperBoundD2 DO
		FOR k := lowerBoundD3 TO upperBoundD3 DO
	
			IF array3D.TryGetElementAsDatatypeByIndex(i, j, k, element) THEN
				elementClone := element.Clone();
				datatypeOperations.AddMemoryCopyOperation(element, elementClone);
				AddOutput(Get3DIndexName(i,j,k), elementClone);
				selfMadeElements.Push(elementClone);
			END_IF
			
		END_FOR
	END_FOR
END_FOR
END_METHOD

METHOD PRIVATE Get1DIndexName : T_MAXSTRING
VAR_INPUT
	Index : DINT;
END_VAR
Get1DIndexName := concat('[',DINT_TO_STRING(Index));
Get1DIndexName := concat(Get1DIndexName,']');
END_METHOD

METHOD PRIVATE Get2DIndexName : T_MAXSTRING
VAR_INPUT
	Index1 : DINT;
	Index2 : DINT;
END_VAR
Get2DIndexName := concat('[',DINT_TO_STRING(Index1));
Get2DIndexName := concat(Get2DIndexName,',');
Get2DIndexName := concat(Get2DIndexName,DINT_TO_STRING(Index2));
Get2DIndexName := concat(Get2DIndexName,']');
END_METHOD

METHOD PRIVATE Get3DIndexName : T_MAXSTRING
VAR_INPUT
	Index1 : DINT;
	Index2 : DINT;
	Index3 : DINT;
END_VAR
Get3DIndexName := concat('[',DINT_TO_STRING(Index1));
Get3DIndexName := concat(Get3DIndexName,',');
Get3DIndexName := concat(Get3DIndexName,DINT_TO_STRING(Index2));
Get3DIndexName := concat(Get3DIndexName,',');
Get3DIndexName := concat(Get3DIndexName,DINT_TO_STRING(Index3));
Get3DIndexName := concat(Get3DIndexName,']');
END_METHOD

METHOD PUBLIC Clone : I_Node
VAR
	pNode : POINTER TO AnyArrayUnbundleNode;
END_VAR
pNode := __NEW(AnyArrayUnbundleNode(ArrayDatatype := in));
Clone := pNode^;
END_METHOD

METHOD PROTECTED OnExecute
VAR
END_VAR
memcpy(out.Address, in.Address, in.Size);
datatypeOperations.Execute();
END_METHOD

END_FUNCTION_BLOCK

// Node/Display/AnyDisplayNode
{attribute 'linkalways'} 
{attribute 'no_explicit_call' := 'This FB is a CLASS and must be accessed using methods or properties'}
{attribute 'enable_dynamic_creation'}
FUNCTION_BLOCK FINAL AnyDisplayNode EXTENDS Node
VAR
	in : I_Datatype;
	display : I_Datatype;
END_VAR

METHOD FB_init : BOOL
VAR_INPUT
	bInitRetains : BOOL; // if TRUE, the retain variables are initialized (warm start / cold start)
	bInCopyCode : BOOL;  // if TRUE, the instance afterwards gets moved into the copy code (online change)
	Datatype : I_Datatype;
END_VAR
THIS^.in := Datatype.Clone();
THIS^.display := Datatype.Clone();

AddInput('in', THIS^.in);
AddContent('display', THIS^.display);
END_METHOD

METHOD FB_exit : BOOL
VAR_INPUT
	bInCopyCode : BOOL; // if TRUE, the exit method is called for exiting an instance that is copied afterwards (online change).
END_VAR
IF bInCopyCode THEN
	RETURN;
END_IF

in.Dispose();
display.Dispose();
END_METHOD

METHOD PUBLIC Clone : I_Node
VAR
	pNode : POINTER TO AnyDisplayNode;
END_VAR
pNode := __NEW(AnyDisplayNode(Datatype := in));
Clone := pNode^;
END_METHOD

METHOD PROTECTED OnExecute
VAR
END_VAR
memcpy(display.Address, in.Address, in.Size);
END_METHOD

END_FUNCTION_BLOCK

// Node/Display/AnyInterfaceDisplayNode
{attribute 'linkalways'} 
{attribute 'no_explicit_call' := 'This FB is a CLASS and must be accessed using methods or properties'}
{attribute 'enable_dynamic_creation'}
FUNCTION_BLOCK FINAL AnyInterfaceDisplayNode EXTENDS Node
VAR
	in : I_InterfaceDatatype;
	display : I_InterfaceDatatype;
END_VAR

METHOD FB_init : BOOL
VAR_INPUT
	bInitRetains : BOOL; // if TRUE, the retain variables are initialized (warm start / cold start)
	bInCopyCode : BOOL;  // if TRUE, the instance afterwards gets moved into the copy code (online change)
	Datatype : I_InterfaceDatatype;
END_VAR
Datatype.Clone().TryResolveAsInterfaceDatatype(THIS^.in);
Datatype.Clone().TryResolveAsInterfaceDatatype(THIS^.display);

AddInput('in', THIS^.in);
AddContent('display', THIS^.display);
END_METHOD

METHOD FB_exit : BOOL
VAR_INPUT
	bInCopyCode : BOOL; // if TRUE, the exit method is called for exiting an instance that is copied afterwards (online change).
END_VAR
IF bInCopyCode THEN
	RETURN;
END_IF

in.Dispose();
display.Dispose();
END_METHOD

METHOD PUBLIC Clone : I_Node
VAR
	pNode : POINTER TO AnyInterfaceDisplayNode;
END_VAR
pNode := __NEW(AnyInterfaceDisplayNode(Datatype := in));
Clone := pNode^;
END_METHOD

METHOD PROTECTED OnExecute
VAR
END_VAR
display.TryCopyContentFrom(in);
END_METHOD

END_FUNCTION_BLOCK

// Node/Literal/AnyLiteralNode
{attribute 'linkalways'} 
{attribute 'no_explicit_call' := 'This FB is a CLASS and must be accessed using methods or properties'}
{attribute 'enable_dynamic_creation'}
FUNCTION_BLOCK FINAL AnyLiteralNode EXTENDS Node
VAR
	value : I_Datatype;
	out : I_Datatype;
	
	// meta
	suppressInputPort : _BOOL(TRUE);
END_VAR

METHOD FB_init : BOOL
VAR_INPUT
	bInitRetains : BOOL; // if TRUE, the retain variables are initialized (warm start / cold start)
	bInCopyCode : BOOL;  // if TRUE, the instance afterwards gets moved into the copy code (online change)
	Datatype : I_Datatype;
END_VAR
THIS^.value := Datatype.Clone();
THIS^.out := Datatype.Clone();

AddParameter('value', THIS^.value)
	.AddMetadata('suppressInput', suppressInputPort); // literals should not use input ports if available. 
	
AddOutput('out', THIS^.out);
END_METHOD

METHOD FB_exit : BOOL
VAR_INPUT
	bInCopyCode : BOOL; // if TRUE, the exit method is called for exiting an instance that is copied afterwards (online change).
END_VAR
IF bInCopyCode THEN
	RETURN;
END_IF

value.Dispose();
out.Dispose();
END_METHOD

METHOD PUBLIC Clone : I_Node
VAR
	pNode : POINTER TO AnyLiteralNode;
END_VAR
pNode := __NEW(AnyLiteralNode(Datatype := value));
Clone := pNode^;
END_METHOD

METHOD PROTECTED OnExecute
VAR
END_VAR
memcpy(out.Address, value.Address, value.Size);
END_METHOD

END_FUNCTION_BLOCK

// Node/Bundle/AnyStructureBundleNode
{attribute 'linkalways'} 
{attribute 'no_explicit_call' := 'This FB is a CLASS and must be accessed using methods or properties'}
{attribute 'enable_dynamic_creation'}
FUNCTION_BLOCK FINAL AnyStructureBundleNode EXTENDS Node
VAR
	in : I_StructuredDatatype;
	out : I_StructuredDatatype;
	datatypeOperations : DatatypeOperations;
	selfMadeMembers : Stack;
END_VAR

METHOD FB_init : BOOL
VAR_INPUT
	bInitRetains : BOOL; // if TRUE, the retain variables are initialized (warm start / cold start)
	bInCopyCode : BOOL;  // if TRUE, the instance afterwards gets moved into the copy code (online change)
	StructuredDatatype : I_StructuredDatatype;
END_VAR
VAR
	enumerator : I_KeyValueForwardEnumerator;
	member : I_Datatype;
	memberAsBit : I_Bit;
	memberAsBool : I_Datatype;
	_bool : pointer to _BOOL;
	memberClone : I_Datatype;
END_VAR
StructuredDatatype.Clone().TryResolveAsStructuredDatatype(out);
AddOutput('out', out);

StructuredDatatype.Clone().TryResolveAsStructuredDatatype(in);
enumerator := in.Members.GetMemberEnumerator();

WHILE enumerator.MoveNext() DO 
	IF enumerator.TryGet(member) THEN
		IF member.TryResolveAs_BIT(memberAsBit) THEN
			// if the element is a _bit then this needs to be treated differently (as you cannot simply memcpy
			// a bit, as it sits next to other data. Instead, a bool is added in it's place.	
			_bool := __NEW(_BOOL(InitialValue := memberAsBit.Value));
			datatypeOperations.AddWriteBoolToBitOperation(_bool^, memberAsBit);
			AddParameter(enumerator.Key, _bool^);
			memberAsBool := _bool^;
			selfMadeMembers.Push(memberAsBool);
		ELSE
			// for all other datatypes,
			memberClone := member.Clone();
			datatypeOperations.AddMemoryCopyOperation(memberClone, member);
			AddParameter(enumerator.key, memberClone);
			selfMadeMembers.Push(memberClone);
		END_IF
	END_IF
END_WHILE

enumerator.Dispose();
END_METHOD

METHOD FB_exit : BOOL
VAR_INPUT
	bInCopyCode : BOOL; // if TRUE, the exit method is called for exiting an instance that is copied afterwards (online change).
END_VAR
VAR
	member : I_Datatype;
END_VAR
IF bInCopyCode THEN
	RETURN;
END_IF

in.Dispose();
out.Dispose();
datatypeOperations.Clear();

WHILE selfMadeMembers.TryPop(member) DO
	IF member <> 0 THEN 
		member.dispose();
	END_IF
END_WHILE
END_METHOD

METHOD PUBLIC Clone : I_Node
VAR
	pNode : POINTER TO AnyStructureBundleNode;
END_VAR
pNode := __NEW(AnyStructureBundleNode(StructuredDatatype := in));
Clone := pNode^;
END_METHOD

METHOD PROTECTED OnExecute
VAR
END_VAR
datatypeOperations.Execute();
memcpy(out.Address, in.Address, in.Size);
END_METHOD

END_FUNCTION_BLOCK

// Node/Unbundle/AnyStructureUnbundleNode
{attribute 'linkalways'} 
{attribute 'no_explicit_call' := 'This FB is a CLASS and must be accessed using methods or properties'}
{attribute 'enable_dynamic_creation'}
FUNCTION_BLOCK FINAL AnyStructureUnbundleNode EXTENDS Node
VAR
	in : I_StructuredDatatype;
	out : I_StructuredDatatype;
	datatypeOperations : DatatypeOperations;
	selfMadeMembers : Stack;
END_VAR

METHOD FB_init : BOOL
VAR_INPUT
	bInitRetains : BOOL; // if TRUE, the retain variables are initialized (warm start / cold start)
	bInCopyCode : BOOL;  // if TRUE, the instance afterwards gets moved into the copy code (online change)
	StructuredDatatype : I_StructuredDatatype;
END_VAR
VAR
	enumerator : I_KeyValueForwardEnumerator;
	member : I_Datatype;
	memberAsBit : I_BIT;
	memberAsBool : I_Datatype;
	_bool : Pointer to _BOOL;
	memberClone : I_Datatype;
END_VAR
StructuredDatatype.Clone().TryResolveAsStructuredDatatype(in);
AddInput('in', in);

StructuredDatatype.Clone().TryResolveAsStructuredDatatype(out);
enumerator := out.Members.GetMemberEnumerator();

WHILE enumerator.MoveNext() DO 
	IF enumerator.TryGet(member) THEN
		IF member.TryResolveAs_BIT(memberAsBit) THEN
			// if the element is a _bit then this needs to be treated differently (as you cannot simply memcpy
			// a bit, as it sits next to other data. Instead, a bool is added in it's place.	
			_bool := __NEW(_BOOL(InitialValue := memberAsBit.Value));
			datatypeOperations.AddWriteBitToBoolOperation(memberAsBit, _bool^);
			AddOutput(enumerator.Key, _bool^);
			memberAsBool := _bool^;
			selfMadeMembers.Push(memberAsBool);
		ELSE
			// for all other datatypes,
			memberClone := member.Clone();
			datatypeOperations.AddMemoryCopyOperation(member, memberClone);
			AddOutput(enumerator.key, memberClone);
			selfMadeMembers.Push(memberClone);
		END_IF		
	END_IF
END_WHILE

enumerator.Dispose();
END_METHOD

METHOD FB_exit : BOOL
VAR_INPUT
	bInCopyCode : BOOL; // if TRUE, the exit method is called for exiting an instance that is copied afterwards (online change).
END_VAR
VAR
	member : I_Datatype;
END_VAR
IF bInCopyCode THEN
	RETURN;
END_IF

in.Dispose();
out.Dispose();
datatypeOperations.Clear();

WHILE selfMadeMembers.TryPop(member) DO
	IF member <> 0 THEN 
		member.dispose();
	END_IF
END_WHILE
END_METHOD

METHOD PUBLIC Clone : I_Node
VAR
	pNode : POINTER TO AnyStructureUnbundleNode;
END_VAR
pNode := __NEW(AnyStructureUnbundleNode(StructuredDatatype := in));
Clone := pNode^;
END_METHOD

METHOD PROTECTED OnExecute
VAR
END_VAR
memcpy(out.Address, in.Address, in.Size);
datatypeOperations.Execute();
END_METHOD

END_FUNCTION_BLOCK

// Graph/Base/Graph
{attribute 'linkalways'} 
{attribute 'no_explicit_call' := 'This FB is a CLASS and must be accessed using methods or properties'}
{attribute 'enable_dynamic_creation'}
FUNCTION_BLOCK Graph EXTENDS Disposable IMPLEMENTS I_Graph
VAR
	nodeFactory : I_NodeFactory;
	_uuid : T_MAXSTRING;	
	eventEmitter : EventEmitter;
	nodeHost : NodeHost(THIS^, eventEmitter);
	inputPortHost : InputPortHost(THIS^, eventEmitter);
	outputPortHost : OutputPortHost(THIS^, eventEmitter);
	parameterHost : ParameterHost(THIS^, eventEmitter);
	contentHost : ContentHost(THIS^, eventEmitter);
	alarmHost : AlarmHost(THIS^, eventEmitter);
	metadataHost : MetadataHost(THIS^, eventEmitter);
	extensionHost : ExtensionHost(THIS^,eventEmitter);
	selfCreatedNodes : Stack;
	nodelinks : NodeLinks;
	
	deserializationFailedAlarm : DeserializationFailedAlarm(THIS^);
	deserializationFailedNodeNotSupportedAlarm : DeserializationFailedNodeNotSupportedAlarm(THIS^);
END_VAR

METHOD FB_init : BOOL
VAR_INPUT
	bInitRetains : BOOL; // if TRUE, the retain variables are initialized (warm start / cold start)
	bInCopyCode : BOOL;  // if TRUE, the instance afterwards gets moved into the copy code (online change)
	NodeFactory : I_NodeFactory;
END_VAR
THIS^.nodeFactory := NodeFactory;
END_METHOD

METHOD FB_exit : BOOL
VAR_INPUT
	bInCopyCode : BOOL; // if TRUE, the exit method is called for exiting an instance that is copied afterwards (online change).
END_VAR
IF bInCopyCode THEN
	RETURN;
END_IF

Clear();
END_METHOD

METHOD PRIVATE DisposeSelfCreatedNodes : BOOL
VAR
	node : I_Node;
END_VAR
WHILE selfCreatedNodes.TryPop(node) DO
	nodeHost.RemoveNode(node);
	node.Dispose();
END_WHILE
END_METHOD

METHOD PRIVATE TryConnectLinksInExecutionOrder : BOOL
VAR_INPUT
END_VAR
VAR
	nodeEnumerator : I_ForwardEnumerator;
	linkEnumerator : I_KeyValueForwardEnumerator;
	nodeId : T_MAXSTRING;
	node : I_Node;
	link : I_NodeLink;
END_VAR
nodeEnumerator := nodes.GetCyclicNodeEnumerator();
linkEnumerator := nodelinks.GetKeyValueEnumerator();

WHILE (nodeEnumerator.MoveNext()) DO
	
	IF nodeEnumerator.TryGet(node) THEN
		nodeId := node.Id;
		linkEnumerator.Reset();
		
		WHILE (linkEnumerator.MoveNext()) DO
	
			IF linkEnumerator.TryGet(link) AND_THEN link.SourceNode.Id = nodeId THEN
				IF NOT link.TryConnect() THEN
					linkEnumerator.Dispose();
					nodeEnumerator.Dispose();
					RETURN;	
				END_IF
			END_IF
		
		END_WHILE

	END_IF

END_WHILE

linkEnumerator.Dispose();
nodeEnumerator.Dispose();
TryConnectLinksInExecutionOrder := TRUE;
END_METHOD

METHOD PUBLIC TryDeserializeNodeLinks : BOOL
VAR_INPUT
	Deserializer : I_Deserializer;
	Feedback : I_DeserializerFeedback;
END_VAR
VAR
	linksDeserializer : I_Deserializer;
	linksEnumerator : I_DeserializerArrayForwardEnumerator;
	linkDeserializer : I_Deserializer;
	linkId : T_MAXSTRING;
	sourceNodeId : T_MAXSTRING;
	sourceName : T_MAXSTRING;
	destinationNodeId : T_MAXSTRING;
	destinationName : T_MAXSTRING;
	sourceNode : I_Node;
	sourcePort : I_OutputPort;
	destinationNode : I_Node;
	destinationPort : I_InputPort;
	destinationParameter : I_Parameter;
	link : I_NodeLink;
END_VAR
linksDeserializer := Deserializer.GetKeyArray('links');
linksEnumerator := linksDeserializer.GetArrayEnumerator();

WHILE linksEnumerator.MoveNext() DO
	
	linkDeserializer := linksEnumerator.Current.GetArray();
	
	IF NOT linkDeserializer.GetElementByIndex(0).TryGetString(linkId, Feedback) THEN
		DeserializationFailedAlarm.Raise('Missing linkid from link');
		linksEnumerator.Dispose();
		RETURN;
	END_IF
	
	IF NOT linkDeserializer.GetElementByIndex(1).TryGetString(sourceNodeId, Feedback) THEN
		DeserializationFailedAlarm.Raise('Missing source node id from link');
		linksEnumerator.Dispose();
		RETURN;
	END_IF
	
	IF NOT linkDeserializer.GetElementByIndex(2).TryGetString(sourceName, Feedback) THEN
		DeserializationFailedAlarm.Raise('Missing source name from link');
		linksEnumerator.Dispose();
		RETURN;
	END_IF
	
	IF NOT linkDeserializer.GetElementByIndex(3).TryGetString(destinationNodeId, Feedback) THEN
		DeserializationFailedAlarm.Raise('Missing destination node id from link');
		linksEnumerator.Dispose();
		RETURN;
	END_IF
	
	IF NOT linkDeserializer.GetElementByIndex(4).TryGetString(destinationName, Feedback) THEN
		DeserializationFailedAlarm.Raise('Missing destination name from link');
		linksEnumerator.Dispose();
		RETURN;
	END_IF
	
	IF NOT nodeHost.TryGetNodeById(sourceNodeId, sourceNode) THEN
		DeserializationFailedAlarm.Raise('Unable to get source node when creating link');
		linksEnumerator.Dispose();
		RETURN;
	END_IF
	
	IF NOT nodeHost.TryGetNodeById(destinationNodeId, destinationNode) THEN
		DeserializationFailedAlarm.Raise('Unable to get destination node when creating link');
		linksEnumerator.Dispose();
		RETURN;
	END_IF
	
	IF NOT sourceNode.OutputPorts.TryGetOutputPortByName(sourceName, sourcePort) THEN
		DeserializationFailedAlarm.Raise('Unable to get source when creating link');
		linksEnumerator.Dispose();
		RETURN;
	END_IF
	
	// first try to find the name in the node input ports, then by node parameters
	IF destinationNode.InputPorts.TryGetInputPortByName(destinationName, destinationPort) THEN
		nodelinks.Create(linkId, sourceNode, sourcePort, destinationNode, destinationPort);
	ELSIF  destinationNode.Parameters.TryGetParameterByName(destinationName, destinationParameter) THEN
		nodelinks.Create(linkId, sourceNode, sourcePort, destinationNode, destinationParameter);
	ELSE
		DeserializationFailedAlarm.Raise('Unable to get destination port when creating link');
		linksEnumerator.Dispose();
		RETURN;
	END_IF
	

END_WHILE

IF NOT TryConnectLinksInExecutionOrder() THEN
	DeserializationFailedAlarm.Raise('Unable to finalise links');
	linksEnumerator.Dispose();
	RETURN;
END_IF

TryDeserializeNodeLinks := TRUE;
linksEnumerator.Dispose();
END_METHOD

METHOD PUBLIC TryDeserializeNodes : BOOL;
VAR_INPUT
	Deserializer : I_Deserializer;
	Feedback : I_DeserializerFeedback;
END_VAR
VAR
	nodeDeserializer : I_Deserializer;
	nodesEnumerator : I_DeserializerArrayForwardEnumerator;
	nodeType : T_MAXSTRING;
	pError : POINTER TO MissingNodePrototypeDeserializationError;
	node : I_Node;
END_VAR
nodeDeserializer := Deserializer.GetKeyArray('nodes');
nodesEnumerator := nodeDeserializer.GetArrayEnumerator();

WHILE nodesEnumerator.MoveNext() DO
	
	IF NOT nodesEnumerator.Current.TryGetKeyString('type',nodeType, Feedback) THEN
		RETURN;
	END_IF
	
	IF NOT nodeFactory.TryCreateNodeByType(nodeType, node) THEN
		pError := __NEW(MissingNodePrototypeDeserializationError(MissingType := nodeType));
		Feedback.LogError(pError^);
		DeserializationFailedNodeNotSupportedAlarm.Raise(nodeType);
		nodesEnumerator.Dispose();
		RETURN;
	END_IF
	
	selfCreatedNodes.Push(node);
	
	IF NOT node.TryDeserializeFrom(nodesEnumerator.Current, Feedback) THEN
		DeserializationFailedAlarm.Raise('Node failed to deserialize');
		nodesEnumerator.Dispose();
		RETURN;
	END_IF
	
	Nodes.AddNode(node);

END_WHILE

TryDeserializeNodes := TRUE;
nodesEnumerator.Dispose();
END_METHOD

METHOD PUBLIC Accept
VAR_INPUT
	Visitor : I_GraphVisitor;
END_VAR
Visitor.VisitGraph(THIS^);
END_METHOD

METHOD PUBLIC AddMetadata : I_HostMetadata
VAR_INPUT
	Name : T_MAXSTRING;
	Data : I_Datatype;
END_VAR
Metadatum.AddDataAsMetadata(Name, Data);
AddMetadata := THIS^;
END_METHOD

PROPERTY PUBLIC Alarms : I_Alarms
GET
Alarms := alarmHost;
END_GET
END_PROPERTY

METHOD PUBLIC Clear
VAR_INPUT
END_VAR
_uuid := '';
nodeLinks.Clear();
DisposeSelfCreatedNodes();
END_METHOD

PROPERTY PUBLIC Contents : I_Contents
GET
Contents := contentHost;
END_GET
END_PROPERTY

PROPERTY PUBLIC Extensions : I_Extensions
GET
Extensions := extensionHost;
END_GET
END_PROPERTY

PROPERTY PUBLIC HasRaisedAlarm : BOOL
GET
HasRaisedAlarm := alarmHost.HasRaisedAlarm;
END_GET
END_PROPERTY

PROPERTY PUBLIC InputPorts : I_InputPorts
GET
InputPorts := inputPortHost;
END_GET
END_PROPERTY

PROPERTY PUBLIC Metadatum : I_Metadatum
GET
Metadatum := metadataHost;
END_GET
END_PROPERTY

PROPERTY PUBLIC Nodes : I_Nodes
GET
Nodes := nodeHost;
END_GET
END_PROPERTY

METHOD PUBLIC OffEvent
VAR_INPUT
	EventName : T_MaxString;
	EventHandler : I_EventHandler;
END_VAR
eventEmitter.OffEvent(EventName, EventHandler);
END_METHOD

METHOD PUBLIC OnceEvent
VAR_INPUT
	EventName : T_MaxString;
	EventHandler : I_EventHandler;
END_VAR
eventEmitter.OnceEvent(EventName, EventHandler);
END_METHOD

METHOD PUBLIC OnEvent
VAR_INPUT
	EventName : T_MaxString;
	EventHandler : I_EventHandler;
END_VAR
eventEmitter.OnEvent(EventName, EventHandler);
END_METHOD

PROPERTY PUBLIC OutputPorts : I_OutputPorts
GET
OutputPorts := outputPortHost;
END_GET
END_PROPERTY

PROPERTY PUBLIC Parameters : I_Parameters
GET
Parameters := parameterHost;
END_GET
END_PROPERTY

METHOD PUBLIC SerializeWith
VAR_INPUT
	Serializer : I_Serializer;
END_VAR
Serializer.StartObject();
Serializer.AddKeyString('uuid',_uuid);
inputPortHost.SerializeWith(Serializer);
outputPortHost.SerializeWith(Serializer);
parameterHost.SerializeWith(Serializer);
contentHost.SerializeWith(Serializer);
alarmHost.SerializeWith(Serializer);
extensionHost.SerializeWith(Serializer);
metadataHost.SerializeWith(Serializer);
nodeHost.SerializeWith(Serializer);
Serializer.EndObject();
END_METHOD

METHOD PUBLIC TryDeserializeFrom : BOOL
VAR_INPUT
	Deserializer : I_Deserializer;
	Feedback : I_DeserializerFeedback;
END_VAR
VAR
	receivedUuid : T_MAXSTRING;
END_VAR
DeserializationFailedNodeNotSupportedAlarm.Clear();
DeserializationFailedAlarm.Clear();

IF NOT parameterHost.TryDeserializeFrom(Deserializer, Feedback) THEN
	RETURN;
END_IF

IF NOT extensionHost.TryDeserializeFrom(Deserializer, Feedback) THEN
	RETURN;
END_IF

IF NOT Deserializer.TryGetKeyString('uuid', receivedUuid, Feedback) THEN
	RETURN;
END_IF

Clear();

IF NOT TryDeserializeNodes(Deserializer, Feedback) THEN 
	RETURN;
END_IF

IF NOT TryDeserializeNodeLinks(Deserializer, Feedback) THEN
	RETURN;
END_IF

_uuid := receivedUuid;
TryDeserializeFrom := TRUE;
END_METHOD

PROPERTY PUBLIC Uuid : T_MAXSTRING
GET
Uuid := _uuid;
END_GET
END_PROPERTY

END_FUNCTION_BLOCK

// Node/Host/NodeHost
{attribute 'linkalways'} 
{attribute 'no_explicit_call' := 'This FB is a CLASS and must be accessed using methods or properties'}
{attribute 'enable_dynamic_creation'}
FUNCTION_BLOCK NodeHost IMPLEMENTS I_Nodes, I_Serializable
VAR
	hostParent : I_HostNodes;
	eventTarget : I_EventTarget;
	allNodes : OrderedDictionary;
	cyclicNodes : LinkedList;
	executeEnumerator : I_ForwardEnumerator;
END_VAR

METHOD FB_init : BOOL
VAR_INPUT
	bInitRetains : BOOL; // if TRUE, the retain variables are initialized (warm start / cold start)
	bInCopyCode : BOOL;  // if TRUE, the instance afterwards gets moved into the copy code (online change)
	Parent : I_HostNodes;
	parentEventTarget : I_EventTarget;
END_VAR
hostParent := Parent;
eventTarget := parentEventTarget;
END_METHOD

METHOD PROTECTED AddCyclicNode
VAR_INPUT
	Node : I_Node;
END_VAR
VAR
	currentPosition : I_LinkedListNode;
	currentNode : I_Node;
END_VAR
IF Node = 0 THEN
	RETURN;
END_IF

// is the list empty?
IF cyclicNodes.First = 0 THEN
	// if so, add our node first and jump out as done.
	cyclicNodes.AddFirst(Node);
	RETURN;
END_IF

// if not empty, then is our node higher priorty than the first in the list. 
cyclicNodes.First.TryGet(currentNode); 
IF currentNode.Order > Node.Order THEN
	// if yes, we are now first, jump out as done. 
	cyclicNodes.AddFirst(Node);
	RETURN;
END_IF

// here, the list has something in it, and we have less priority than the node in first place.

// get the last node in the list and remember this as "currentPosition" 
currentPosition := cyclicNodes.Last;

WHILE (TRUE) DO
	
	currentPosition.TryGet(currentNode); 
	// is the current position higer priority than our node?
	IF currentNode.Order <= Node.Order THEN
		// if so, then we go after, jump out as we are done. 
		cyclicNodes.AddAfter(currentPosition, Node);
		RETURN;
	END_IF
	
	// move one up the list towards the top and try again.
	currentPosition := currentPosition.Previous;

END_WHILE
END_METHOD

METHOD PROTECTED EmitOnNodeAddedEvent
VAR_INPUT
	Node : I_Node;
END_VAR
VAR
	nodeAddedEvent : NodeAddedEvent(Target := Node);
END_VAR
IF eventTarget = 0 THEN
	RETURN;
END_IF

eventTarget.Emit('OnNodeAdded', nodeAddedEvent);
END_METHOD

METHOD PUBLIC Accept
VAR_INPUT
	Visitor : I_NodeVisitor;
END_VAR
VAR
	enumerator : I_ForwardEnumerator;
	node : I_Node;
END_VAR
enumerator := allNodes.GetEnumerator();

WHILE (enumerator.MoveNext()) DO
	
	IF enumerator.TryGet(node) THEN
		node.Accept(Visitor);
	END_IF

END_WHILE

enumerator.Dispose();
END_METHOD

METHOD PUBLIC AddNode
VAR_INPUT
	Node : I_Node;
END_VAR
allNodes.AddOrUpdate(Node.id, Node);

IF Node.IsCyclicMode THEN
	AddCyclicNode(Node);
END_IF

EmitOnNodeAddedEvent(Node);
END_METHOD

METHOD PUBLIC GetAllNodeEnumerator : I_KeyValueForwardEnumerator
VAR_INPUT
END_VAR
GetAllNodeEnumerator := allNodes.GetKeyValueEnumerator();
END_METHOD

METHOD PUBLIC GetCyclicNodeEnumerator : I_ForwardEnumerator
VAR_INPUT
END_VAR
GetCyclicNodeEnumerator := cyclicNodes.GetEnumerator();
END_METHOD

PROPERTY PUBLIC HasNodes : BOOL
GET
//HasNodes := NOT nodes.IsEmpty;
HasNodes := NOT allNodes.IsEmpty OR NOT cyclicNodes.IsEmpty;
END_GET
END_PROPERTY

METHOD PUBLIC RemoveNode
VAR_INPUT
	Node : I_Node;
END_VAR
allNodes.Remove(Node.Id);
cyclicNodes.Remove(Node);
END_METHOD

METHOD PUBLIC SerializeWith
VAR_INPUT
	Serializer : I_Serializer;
END_VAR
VAR
	enumerator : I_ForwardEnumerator;
	node : I_Node;
END_VAR
IF allNodes.Count = 0 THEN
	RETURN;
END_IF

Serializer.AddKey('nodes');
Serializer.StartArray();

enumerator := allNodes.GetEnumerator();

WHILE enumerator.MoveNext() DO
	IF enumerator.TryGet(node) THEN
		node.SerializeWith(Serializer);
	END_IF
END_WHILE

Serializer.EndArray();
enumerator.Dispose();
END_METHOD

METHOD PUBLIC TryDeserializeFrom : BOOL
VAR_INPUT
	Deserializer : I_Deserializer;
	Feedback : I_DeserializerFeedback;
END_VAR
VAR
	nodeDeserializer : I_Deserializer;
	nodesEnumerator : I_DeserializerArrayForwardEnumerator;
	nodeId : T_MAXSTRING;
	node : I_Node;
END_VAR
nodeDeserializer := Deserializer.GetKeyArray('nodes');
nodesEnumerator := nodeDeserializer.GetArrayEnumerator();

WHILE nodesEnumerator.MoveNext() DO
	
	IF NOT nodesEnumerator.Current.TryGetKeyString('id', nodeId, Feedback) THEN
		CONTINUE;
	END_IF
	
	IF NOT TryGetNodeById(nodeId, node)THEN
		CONTINUE;
	END_IF
	
	node.TryDeserializeFrom(nodesEnumerator.Current, Feedback);

END_WHILE

nodesEnumerator.Dispose();
END_METHOD

METHOD PUBLIC TryGetNodeById : BOOL
VAR_INPUT
	Id : T_MAXSTRING;
	Destination : REFERENCE TO I_Node;
END_VAR
VAR
	node : I_Node;
END_VAR
IF NOT allNodes.TryGetValue(Id, node) THEN
	RETURN;
END_IF

Destination := node;
TryGetNodeById := TRUE;
END_METHOD

END_FUNCTION_BLOCK

// Node/Events/NodeAddedEvent
{attribute 'linkalways'} 
{attribute 'no_explicit_call' := 'This FB is a CLASS and must be accessed using methods or properties'}
{attribute 'enable_dynamic_creation'}
FUNCTION_BLOCK NodeAddedEvent EXTENDS Disposable IMPLEMENTS I_NodeAddedEvent
VAR
	_target : I_Node;
END_VAR

METHOD FB_init : BOOL
VAR_INPUT
	bInitRetains : BOOL; // if TRUE, the retain variables are initialized (warm start / cold start)
	bInCopyCode : BOOL;  // if TRUE, the instance afterwards gets moved into the copy code (online change)
	Target : I_Node;
END_VAR
THIS^._target := Target;
END_METHOD

PROPERTY PUBLIC Target : I_Node
GET
Target := _target;
END_GET
END_PROPERTY

END_FUNCTION_BLOCK

// Node/Events/I_NodeAddedEvent
INTERFACE I_NodeAddedEvent EXTENDS I_Event

PROPERTY PUBLIC Target : I_Node
GET
END_GET
END_PROPERTY

END_INTERFACE

// Link/Collection/NodeLinks
{attribute 'linkalways'} 
{attribute 'no_explicit_call' := 'This FB is a CLASS and must be accessed using methods or properties'}
{attribute 'enable_dynamic_creation'}
FUNCTION_BLOCK NodeLinks EXTENDS disposable IMPLEMENTS I_NodeLinks
VAR
	links : OrderedDictionary;
END_VAR

METHOD FB_exit : BOOL
VAR_INPUT
	bInCopyCode : BOOL; // if TRUE, the exit method is called for exiting an instance that is copied afterwards (online change).
END_VAR
IF bInCopyCode THEN
	RETURN;
END_IF

Clear();
END_METHOD

METHOD PRIVATE CreateNewLink : I_NodeLink
VAR_INPUT
	LinkId : T_MAXSTRING;
	LinkSourceNode : I_Node;
	LinkSource : I_LinkSource;
	LinkDestinationNode : I_Node;
	LinkDestination : I_LinkDestination;
END_VAR
VAR
	pLink : POINTER TO Link;
END_VAR
pLink := __NEW(
	Link(
		Id := LinkId, 
		SourceNode := LinkSourceNode,
		Source := LinkSource,
		DestinationNode := LinkDestinationNode,
		Destination := LinkDestination
	)
);

CreateNewLink := pLink^;
END_METHOD

METHOD PUBLIC Clear
VAR_INPUT
END_VAR
VAR
	enumerator : I_ForwardEnumerator;
	link : I_NodeLink;
END_VAR
enumerator := links.GetEnumerator();

WHILE (enumerator.MoveNext()) DO
	
	IF enumerator.TryGet(link) THEN
		link.Dispose();
	END_IF

END_WHILE

enumerator.Dispose();
links.Clear();
END_METHOD

METHOD PUBLIC Create : I_NodeLink
VAR_INPUT
	LinkId : T_MAXSTRING;
	LinkSourceNode : I_Node;
	LinkSource : I_LinkSource;
	LinkDestinationNode : I_Node;
	LinkDestination : I_LinkDestination;
END_VAR
VAR
	link : I_NodeLink;
END_VAR
link := CreateNewLink(
	LinkId, 
	LinkSourceNode,
	LinkSource,
	LinkDestinationNode,
	LinkDestination
);

links.AddOrUpdate(link.Id, link);
Create := link;
END_METHOD

METHOD PUBLIC DisconnectAll
VAR_INPUT
END_VAR
VAR
	enumerator : I_ForwardEnumerator;
	link : I_NodeLink;
END_VAR
enumerator := links.GetEnumerator();

WHILE (enumerator.MoveNext()) DO
	
	IF enumerator.TryGet(link) THEN
		link.Disconnect();
	END_IF

END_WHILE

enumerator.Dispose();
END_METHOD

METHOD PUBLIC GetKeyValueEnumerator : I_KeyValueForwardEnumerator
VAR_INPUT
END_VAR
GetKeyValueEnumerator := links.GetKeyValueEnumerator();
END_METHOD

METHOD PUBLIC TryGetLinkById : BOOL
VAR_INPUT
	Id : T_MAXSTRING;
	Destination : REFERENCE TO I_NodeLink;
END_VAR
VAR
	link : I_NodeLink;
END_VAR
IF NOT links.TryGetValue(Id, link) THEN
	RETURN;
END_IF

Destination := link;
TryGetLinkById := TRUE;
END_METHOD

END_FUNCTION_BLOCK

// Link/Interface/I_NodeLinks
INTERFACE I_NodeLinks EXTENDS I_Disposable

METHOD PUBLIC Clear
VAR_INPUT
END_VAR
END_METHOD

METHOD PUBLIC Create : I_NodeLink
VAR_INPUT
	LinkId : T_MAXSTRING;
	LinkSourceNode : I_Node;
	LinkSource : I_LinkSource;
	LinkDestinationNode : I_Node;
	LinkDestination : I_LinkDestination;
END_VAR
END_METHOD

METHOD PUBLIC DisconnectAll
VAR_INPUT
END_VAR
END_METHOD

METHOD PUBLIC GetKeyValueEnumerator : I_KeyValueForwardEnumerator
VAR_INPUT
END_VAR
END_METHOD

METHOD PUBLIC TryGetLinkById : BOOL
VAR_INPUT
	Id : T_MAXSTRING;
	Destination : REFERENCE TO I_NodeLink;
END_VAR
END_METHOD

END_INTERFACE

// Link/Interface/I_NodeLink
INTERFACE I_NodeLink EXTENDS I_Disposable

PROPERTY PUBLIC Destination : I_LinkDestination
GET
END_GET
END_PROPERTY

PROPERTY PUBLIC DestinationNode : I_Node
GET
END_GET
END_PROPERTY

METHOD PUBLIC Disconnect
VAR_INPUT
END_VAR
END_METHOD

PROPERTY PUBLIC Id : T_MAXSTRING
GET
END_GET
END_PROPERTY

PROPERTY PUBLIC Source : I_LinkSource
GET
END_GET
END_PROPERTY

PROPERTY PUBLIC SourceNode : I_Node
GET
END_GET
END_PROPERTY

METHOD PUBLIC TryConnect : BOOL;
VAR_INPUT
END_VAR
END_METHOD

END_INTERFACE

// Link/Link
{attribute 'linkalways'} 
{attribute 'no_explicit_call' := 'This FB is a CLASS and must be accessed using methods or properties'}
{attribute 'enable_dynamic_creation'}
FUNCTION_BLOCK Link EXTENDS Disposable IMPLEMENTS I_NodeLink
VAR
	_id : T_MAXSTRING;
	_sourceNode : I_Node;
	_source : I_LinkSource;
	_destinationNode : I_Node;
	_destination : I_LinkDestination;
END_VAR

METHOD FB_init : BOOL
VAR_INPUT
	bInitRetains : BOOL; // if TRUE, the retain variables are initialized (warm start / cold start)
	bInCopyCode : BOOL;  // if TRUE, the instance afterwards gets moved into the copy code (online change)
	Id : T_MAXSTRING;
	SourceNode : I_Node;
	Source : I_LinkSource;
	DestinationNode : I_Node;
	Destination : I_LinkDestination;
END_VAR
_id := Id;
_sourceNode := SourceNode;
_source := Source;
_destinationNode := DestinationNode;
_destination := Destination;
END_METHOD

METHOD FB_exit : BOOL
VAR_INPUT
	bInCopyCode : BOOL; // if TRUE, the exit method is called for exiting an instance that is copied afterwards (online change).
END_VAR
IF bInCopyCode THEN
	RETURN;
END_IF

Disconnect();
END_METHOD

PROPERTY PUBLIC Destination : I_LinkDestination
GET
Destination := _destination;
END_GET
END_PROPERTY

PROPERTY PUBLIC DestinationNode : I_Node
GET
DestinationNode := _destinationNode;
END_GET
END_PROPERTY

METHOD PUBLIC Disconnect
VAR_INPUT
END_VAR
IF _source = 0 THEN
	RETURN;
END_IF

IF _destination = 0 THEN
	RETURN;
END_IF

_destination.Disconnect();
END_METHOD

PROPERTY PUBLIC Id : T_MAXSTRING
GET
Id := _id;
END_GET
END_PROPERTY

PROPERTY PUBLIC Source : I_LinkSource
GET
Source := _source;
END_GET
END_PROPERTY

PROPERTY PUBLIC SourceNode : I_Node
GET
SourceNode := _sourceNode;
END_GET
END_PROPERTY

METHOD PUBLIC TryConnect : BOOL;
VAR_INPUT
END_VAR
IF _source = 0 THEN
	RETURN;
END_IF

IF _destination = 0 THEN
	RETURN;
END_IF

TryConnect := _destination.TryConnectTo(_source);
END_METHOD

END_FUNCTION_BLOCK

// Errors/MissingNodePrototypeDeserializationError
{attribute 'linkalways'} 
{attribute 'no_explicit_call' := 'This FB is a CLASS and must be accessed using methods or properties'}
{attribute 'enable_dynamic_creation'}
FUNCTION_BLOCK MissingNodePrototypeDeserializationError EXTENDS Error
VAR
	nodeType : T_MAXSTRING;
END_VAR

METHOD FB_init : BOOL
VAR_INPUT
	bInitRetains : BOOL; // if TRUE, the retain variables are initialized (warm start / cold start)
	bInCopyCode : BOOL;  // if TRUE, the instance afterwards gets moved into the copy code (online change)
	MissingType : T_MAXSTRING;
END_VAR
nodeType := MissingType;
END_METHOD

PROPERTY PUBLIC ErrorType : T_MAXSTRING
GET
ErrorType := 'MISSING_NODE_PROTOTYPE_DESERIALIZATION_ERROR';
END_GET
END_PROPERTY

PROPERTY PUBLIC Message : T_MAXSTRING
GET
Message := CONCAT('Deserialization Failed, Missing Node Prototype : ',nodeType);
END_GET
END_PROPERTY

END_FUNCTION_BLOCK

// GraphRuntime/Interface/I_GraphRuntimeCollection
INTERFACE I_GraphRuntimeCollection

METHOD PUBLIC Accept
VAR_INPUT
	Visitor : I_GraphRuntimeVisitor;
END_VAR
END_METHOD

METHOD PUBLIC AddDefaultRuntime
VAR_INPUT
	GraphRuntime : I_GraphRuntime;
END_VAR
END_METHOD

METHOD PUBLIC AddRuntimeById
VAR_INPUT
	Id : T_MAXSTRING;
	GraphRuntime : I_GraphRuntime;
END_VAR
END_METHOD

METHOD PUBLIC RemoveDefaultRuntime
VAR_INPUT
END_VAR
END_METHOD

METHOD PUBLIC RemoveRuntimeById
VAR_INPUT
	Id : T_MAXSTRING;
END_VAR
END_METHOD

METHOD PUBLIC TryGetDefaultRuntime : BOOL
VAR_INPUT
	Destination : REFERENCE TO I_GraphRuntime;
END_VAR
END_METHOD

METHOD PUBLIC TryGetRuntimeById : BOOL
VAR_INPUT
	Id : T_MAXSTRING;
	Destination : REFERENCE TO I_GraphRuntime;
END_VAR
END_METHOD

END_INTERFACE

// Visitors/Interfaces/I_GraphRuntimeVisitor
INTERFACE I_GraphRuntimeVisitor

METHOD VisitGraphRuntime
VAR_INPUT
	VisitingGraphRuntime : I_GraphRuntime;
END_VAR
END_METHOD

END_INTERFACE

// GraphRuntime/Interface/I_GraphRuntime
INTERFACE I_GraphRuntime Extends I_EventEmitter, I_HostGraphInstances

METHOD PUBLIC Accept
VAR_INPUT
	Visitor : I_GraphRuntimeVisitor;
END_VAR
END_METHOD

METHOD PUBLIC AddNewDefaultGraphInstance : I_GraphInstance
VAR_INPUT
	Graph : I_Graph;
END_VAR
END_METHOD

METHOD PUBLIC AddNewGraphInstance : I_GraphInstance
VAR_INPUT
	InstanceId : T_MAXSTRING;
	Graph : I_Graph;
END_VAR
END_METHOD

METHOD PUBLIC DisposeAllInstances
END_METHOD

METHOD PUBLIC DisposeDefaultGraphInstance
END_METHOD

METHOD PUBLIC DisposeGraphInstance
VAR_INPUT
	InstanceId : T_MAXSTRING;
END_VAR
END_METHOD

PROPERTY PUBLIC Id : T_MAXSTRING
GET
END_GET
END_PROPERTY

METHOD PUBLIC TryGetDefaultGraphInstance : BOOL
VAR_INPUT
	Destination : REFERENCE TO I_GraphInstance;
END_VAR
END_METHOD

METHOD PUBLIC TryGetGraphInstance : BOOL
VAR_INPUT
	InstanceId : T_MAXSTRING;
	Destination : REFERENCE TO I_GraphInstance;
END_VAR
END_METHOD

END_INTERFACE

// GraphInstance/Interface/I_HostGraphInstances
INTERFACE I_HostGraphInstances

PROPERTY GraphInstances : I_GraphInstanceHost
GET
END_GET
END_PROPERTY

END_INTERFACE

// GraphInstance/Interface/I_GraphInstanceHost
INTERFACE I_GraphInstanceHost

METHOD PUBLIC Accept
VAR_INPUT
	visitor : I_GraphInstanceVisitor;
END_VAR
END_METHOD

END_INTERFACE

// Visitors/Interfaces/I_GraphInstanceVisitor
INTERFACE I_GraphInstanceVisitor

METHOD VisitGraphInstance
VAR_INPUT
	VisitingGraphInstance : I_GraphInstance;
END_VAR
END_METHOD

END_INTERFACE

// GraphInstance/Interface/I_GraphInstance
INTERFACE I_GraphInstance EXTENDS I_Disposable, I_Serializable

METHOD PUBLIC Accept
VAR_INPUT
	Visitor : I_GraphInstanceVisitor;
END_VAR
END_METHOD

PROPERTY PUBLIC CycleCount : UDINT
GET
END_GET
END_PROPERTY

METHOD PUBLIC CyclicCall
VAR_INPUT
END_VAR
END_METHOD

PROPERTY PUBLIC Graph : I_Graph
GET
END_GET
END_PROPERTY

PROPERTY PUBLIC Id : T_MAXSTRING
GET
END_GET
END_PROPERTY

PROPERTY PUBLIC IsEndOfCycle : BOOL
GET
END_GET
END_PROPERTY

PROPERTY PUBLIC IsRunning : BOOL
GET
END_GET
END_PROPERTY

PROPERTY PUBLIC IsStopped : BOOL
GET
END_GET
END_PROPERTY

METHOD Start
VAR_INPUT
END_VAR
END_METHOD

METHOD Stop
VAR_INPUT
END_VAR
END_METHOD

END_INTERFACE

// GraphRuntime/GraphRuntime
{attribute 'linkalways'} 
{attribute 'no_explicit_call' := 'This FB is a CLASS and must be accessed using methods or properties'}
{attribute 'enable_dynamic_creation'}
FUNCTION_BLOCK GraphRuntime IMPLEMENTS I_GraphRuntime, I_HostGraphInstances, I_EventEmitter
VAR
	cyclicGraphExecutionStrategyProvider : CyclicGraphExecutionStrategyProvider;
	defaultGraphExecutionStrategyProvider : I_GraphExecutionStrategyProvider := cyclicGraphExecutionStrategyProvider;
	_id : T_MAXSTRING;
	eventEmitter : EventEmitter;
	graphInstanceHost : GraphInstanceHost(THIS^, eventEmitter);
END_VAR

METHOD FB_init : BOOL
VAR_INPUT
	bInitRetains : BOOL; // if TRUE, the retain variables are initialized (warm start / cold start)
	bInCopyCode : BOOL;  // if TRUE, the instance afterwards gets moved into the copy code (online change)
	Id : T_MAXSTRING;
END_VAR
THIS^._id := Id;
END_METHOD

METHOD PUBLIC Accept
VAR_INPUT
	Visitor : I_GraphRuntimeVisitor;
END_VAR
Visitor.VisitGraphRuntime(THIS^);
END_METHOD

METHOD PUBLIC AddNewDefaultGraphInstance : I_GraphInstance
VAR_INPUT
	Graph : I_Graph;
END_VAR
AddNewDefaultGraphInstance := graphInstanceHost.AddNewDefaultGraphInstance(Graph, defaultGraphExecutionStrategyProvider);
END_METHOD

METHOD PUBLIC AddNewGraphInstance : I_GraphInstance
VAR_INPUT
	InstanceId : T_MAXSTRING;
	Graph : I_Graph;
END_VAR
AddNewGraphInstance := graphInstanceHost.AddNewGraphInstance(InstanceId, Graph, defaultGraphExecutionStrategyProvider);
END_METHOD

METHOD PUBLIC ChangeDefaultExecutionStrategy : BOOL
VAR_INPUT
	GraphExecutionStrategyProvider : I_GraphExecutionStrategyProvider;
END_VAR
IF GraphExecutionStrategyProvider = 0 THEN
	RETURN;
END_IF

defaultGraphExecutionStrategyProvider := GraphExecutionStrategyProvider;
END_METHOD

METHOD PUBLIC CyclicCall
VAR_INPUT
END_VAR
graphInstanceHost.CyclicCall();
END_METHOD

METHOD PUBLIC DisposeAllInstances
VAR
	graphInstance : I_GraphInstance;
END_VAR
graphInstanceHost.DisposeAll();
END_METHOD

METHOD PUBLIC DisposeDefaultGraphInstance
graphInstanceHost.DisposeDefaultGraphInstance();
END_METHOD

METHOD PUBLIC DisposeGraphInstance
VAR_INPUT
	InstanceId : T_MAXSTRING;
END_VAR
graphInstanceHost.DisposeGraphInstance(InstanceId);
END_METHOD

PROPERTY PUBLIC GraphInstances : I_GraphInstanceHost
GET
GraphInstances := graphInstanceHost;
END_GET
END_PROPERTY

PROPERTY PUBLIC Id : T_MAXSTRING
GET
Id := _id;
END_GET
END_PROPERTY

METHOD PUBLIC OffEvent
VAR_INPUT
	EventName : T_MaxString;
	EventHandler : I_EventHandler;
END_VAR
eventEmitter.OffEvent(EventName, EventHandler);
END_METHOD

METHOD PUBLIC OnceEvent
VAR_INPUT
	EventName : T_MaxString;
	EventHandler : I_EventHandler;
END_VAR
eventEmitter.OnceEvent(EventName, EventHandler);
END_METHOD

METHOD PUBLIC OnEvent
VAR_INPUT
	EventName : T_MaxString;
	EventHandler : I_EventHandler;
END_VAR
eventEmitter.OnEvent(EventName, EventHandler);
END_METHOD

METHOD PUBLIC TryGetDefaultGraphInstance : BOOL
VAR_INPUT
	Destination : REFERENCE TO I_GraphInstance;
END_VAR
TryGetDefaultGraphInstance := graphInstanceHost.TryGetDefaultGraphInstance(Destination);
END_METHOD

METHOD PUBLIC TryGetGraphInstance : BOOL
VAR_INPUT
	InstanceId : T_MAXSTRING;
	Destination : REFERENCE TO I_GraphInstance;
END_VAR
TryGetGraphInstance := graphInstanceHost.TryGetGraphInstance(InstanceId, Destination);
END_METHOD

END_FUNCTION_BLOCK

// GraphExecutionStrategy/Cyclic/CyclicGraphExecutionStrategyProvider
{attribute 'linkalways'} 
{attribute 'no_explicit_call' := 'This FB is a CLASS and must be accessed using methods or properties'}
{attribute 'enable_dynamic_creation'}
FUNCTION_BLOCK CyclicGraphExecutionStrategyProvider EXTENDS Disposable IMPLEMENTS I_GraphExecutionStrategyProvider
VAR
END_VAR

METHOD Create : I_GraphExecutionStrategy
VAR_INPUT
	TargetGraph : I_Graph;
END_VAR
VAR
	pGraphExecutionStrategy : POINTER TO CyclicGraphExecutionStrategy;
END_VAR
pGraphExecutionStrategy := __NEW(CyclicGraphExecutionStrategy(ParentGraph := TargetGraph));
Create := pGraphExecutionStrategy^;
END_METHOD

END_FUNCTION_BLOCK

// GraphExecutionStrategy/Interface/I_GraphExecutionStrategyProvider
INTERFACE I_GraphExecutionStrategyProvider

METHOD Create : I_GraphExecutionStrategy
VAR_INPUT
	TargetGraph : I_Graph;
END_VAR
END_METHOD

END_INTERFACE

// GraphExecutionStrategy/Interface/I_GraphExecutionStrategy
INTERFACE I_GraphExecutionStrategy EXTENDS I_Disposable, I_Serializable

METHOD PUBLIC Accept
VAR_INPUT
	visitor : I_GraphExecutionEngineVisitor;
END_VAR
END_METHOD

PROPERTY PUBLIC CycleCount : UDINT
GET
END_GET
END_PROPERTY

METHOD PUBLIC CyclicCall
END_METHOD

PROPERTY PUBLIC IsEndOfCycle : BOOL
GET
END_GET
END_PROPERTY

PROPERTY PUBLIC IsRunning : BOOL
GET
END_GET
END_PROPERTY

PROPERTY PUBLIC IsStopped : BOOL
GET
END_GET
END_PROPERTY

METHOD PUBLIC SerializeWith
VAR_INPUT
	Serializer : I_Serializer;
END_VAR
END_METHOD

METHOD PUBLIC Start
VAR_INPUT
END_VAR
END_METHOD

METHOD PUBLIC Stop
VAR_INPUT
END_VAR
END_METHOD

END_INTERFACE

// Visitors/Interfaces/I_GraphExecutionEngineVisitor
INTERFACE I_GraphExecutionEngineVisitor

METHOD VisitGraphExecutionEngine
VAR_INPUT
	VisitingGraph : I_GraphExecutionStrategy;
END_VAR
END_METHOD

END_INTERFACE

// GraphExecutionStrategy/Cyclic/CyclicGraphExecutionStrategy
{attribute 'linkalways'} 
{attribute 'no_explicit_call' := 'This FB is a CLASS and must be accessed using methods or properties'}
{attribute 'enable_dynamic_creation'}
FUNCTION_BLOCK CyclicGraphExecutionStrategy EXTENDS Disposable IMPLEMENTS I_GraphExecutionStrategy
VAR
	parentGraph : I_Graph;
	state : (UNINITIALIZED, STOP, START);
	cyclicNodeEnumerator : I_ForwardEnumerator;
	cycleCounter : UDINT;
	endOfCycle : BOOL;
END_VAR

METHOD FB_init : BOOL
VAR_INPUT
	bInitRetains : BOOL; // if TRUE, the retain variables are initialized (warm start / cold start)
	bInCopyCode : BOOL;  // if TRUE, the instance afterwards gets moved into the copy code (online change)
	ParentGraph : I_Graph;
END_VAR
IF parentGraph = 0 THEN
	RETURN;
END_IF

Initialize(ParentGraph);
END_METHOD

METHOD FB_exit : BOOL
VAR_INPUT
	bInCopyCode : BOOL; // if TRUE, the exit method is called for exiting an instance that is copied afterwards (online change).
END_VAR
IF bInCopyCode THEN
	RETURN;
END_IF

IF cyclicNodeEnumerator <> 0 THEN
	cyclicNodeEnumerator.Dispose();
	cyclicNodeEnumerator := 0;
END_IF
END_METHOD

METHOD PRIVATE CycleComplete
VAR_INPUT
END_VAR
cycleCounter := cycleCounter + 1;
endOfCycle := TRUE;
END_METHOD

METHOD PRIVATE CycleStart
VAR_INPUT
END_VAR
endOfCycle := FALSE;
END_METHOD

METHOD PRIVATE GetNewEnumerator
VAR_INPUT
END_VAR
IF cyclicNodeEnumerator <> 0 THEN
	cyclicNodeEnumerator.Dispose();
	cyclicNodeEnumerator := 0;
END_IF

cyclicNodeEnumerator := parentGraph.Nodes.GetCyclicNodeEnumerator();
END_METHOD

METHOD PUBLIC Initialize
VAR_INPUT
	Graph : I_Graph;
END_VAR
parentGraph := Graph;
GetNewEnumerator();
state := STOP;
END_METHOD

METHOD PUBLIC Accept
VAR_INPUT
	visitor : I_GraphExecutionEngineVisitor;
END_VAR
Visitor.VisitGraphExecutionEngine(THIS^);
END_METHOD

PROPERTY PUBLIC CycleCount : UDINT
GET
CycleCount := CycleCounter;
END_GET
END_PROPERTY

METHOD PUBLIC CyclicCall
VAR
	node : I_Node;
END_VAR
IF state = UNINITIALIZED THEN
	RETURN;
END_IF

IF state = STOP THEN
	RETURN;
END_IF

IF NOT cyclicNodeEnumerator.IsValid THEN
	GetNewEnumerator();
ELSE
	cyclicNodeEnumerator.Reset();
END_IF

CycleStart();

WHILE cyclicNodeEnumerator.MoveNext() DO
	IF cyclicNodeEnumerator.TryGet(node) THEN
		node.Execute();
	END_IF
END_WHILE

CycleComplete();
END_METHOD

PROPERTY PUBLIC IsEndOfCycle : BOOL
GET
IsEndOfCycle := endOfCycle;
END_GET
END_PROPERTY

PROPERTY PUBLIC IsRunning : BOOL
GET
IsRunning := state = START;
END_GET
END_PROPERTY

PROPERTY PUBLIC IsStopped : BOOL
GET
IsStopped := state = STOP OR state = UNINITIALIZED;
END_GET
END_PROPERTY

METHOD PUBLIC SerializeWith
VAR_INPUT
	Serializer : I_Serializer;
END_VAR
// to do, serialize the running state of the graph
END_METHOD

METHOD PUBLIC Start
VAR_INPUT
END_VAR
IF state = UNINITIALIZED THEN
	RETURN;
END_IF

state := START;
END_METHOD

METHOD PUBLIC Stop
VAR_INPUT
END_VAR
IF state = UNINITIALIZED THEN
	RETURN;
END_IF

state := STOP;
END_METHOD

END_FUNCTION_BLOCK

// GraphInstance/Host/GraphInstanceHost
{attribute 'linkalways'} 
{attribute 'no_explicit_call' := 'This FB is a CLASS and must be accessed using methods or properties'}
{attribute 'enable_dynamic_creation'}
FUNCTION_BLOCK GraphInstanceHost IMPLEMENTS I_GraphInstanceHost, I_Serializable
VAR
	hostParent : I_HostGraphInstances;
	eventTarget : I_EventTarget;
	graphInstances : OrderedDictionary;	
	enumerator : I_ForwardEnumerator;
END_VAR
VAR CONSTANT
	DEFAULT_ID : T_MAXSTRING := 'default';
END_VAR

METHOD FB_init : BOOL
VAR_INPUT
	bInitRetains : BOOL; // if TRUE, the retain variables are initialized (warm start / cold start)
	bInCopyCode : BOOL;  // if TRUE, the instance afterwards gets moved into the copy code (online change)
	Parent : I_HostGraphInstances;
	ParentEventTarget : I_EventTarget;
END_VAR
hostParent := Parent;
eventTarget := parentEventTarget;
GetNewEnumerator();
END_METHOD

METHOD FB_exit : BOOL
VAR_INPUT
	bInCopyCode : BOOL; // if TRUE, the exit method is called for exiting an instance that is copied afterwards (online change).
END_VAR
IF bInCopyCode THEN
	RETURN;
END_IF

DisposeAll();
DisposeEnumerator();
END_METHOD

METHOD PRIVATE DisposeEnumerator
VAR_INPUT
END_VAR
IF enumerator = 0 THEN
	RETURN;
END_IF

enumerator.Dispose();
enumerator := 0;
END_METHOD

METHOD PRIVATE GetNewEnumerator
VAR_INPUT
END_VAR
IF enumerator <> 0 THEN
	enumerator.Dispose();
	enumerator := 0;
END_IF

enumerator := graphInstances.GetEnumerator();
END_METHOD

METHOD PUBLIC CreateNewGraphInstance : I_GraphInstance
VAR_INPUT
	InstanceId : T_MAXSTRING;
	Graph : I_Graph;
	InstanceExecutionStrategyProvider : I_GraphExecutionStrategyProvider;
END_VAR
VAR
	pGraphInstance : POINTER TO GraphInstance;
END_VAR
pGraphInstance := __NEW(GraphInstance(Id := InstanceId, TargetGraph := Graph, ExecutionStrategyProvider := InstanceExecutionStrategyProvider));
CreateNewGraphInstance := pGraphInstance^;
END_METHOD

METHOD PROTECTED EmitOnGraphInstanceAddedEvent
VAR_INPUT
	GraphInstance : I_GraphInstance;
END_VAR
VAR
	graphInstanceAddedEvent : GraphInstanceAddedEvent(Target := GraphInstance);
END_VAR
IF eventTarget = 0 THEN
	RETURN;
END_IF

eventTarget.Emit('OnGraphInstanceAdded', graphInstanceAddedEvent);
END_METHOD

METHOD PUBLIC Accept
VAR_INPUT
	visitor : I_GraphInstanceVisitor;
END_VAR
VAR
	graphInstance : I_GraphInstance;
END_VAR
IF NOT enumerator.IsValid THEN
	GetNewEnumerator();
ELSE
	enumerator.Reset();
END_IF

WHILE (enumerator.MoveNext()) DO
	
	IF enumerator.TryGet(graphInstance) THEN
		graphInstance.Accept(Visitor);
	END_IF

END_WHILE
END_METHOD

METHOD PUBLIC AddNewDefaultGraphInstance : I_GraphInstance
VAR_INPUT
	Graph : I_Graph;
	InstanceExecutionStrategyProvider : I_GraphExecutionStrategyProvider;
END_VAR
AddNewDefaultGraphInstance := AddNewGraphInstance(DEFAULT_ID, Graph, InstanceExecutionStrategyProvider);
END_METHOD

METHOD PUBLIC AddNewGraphInstance : I_GraphInstance
VAR_INPUT
	InstanceId : T_MAXSTRING;
	Graph : I_Graph;
	InstanceExecutionStrategyProvider : I_GraphExecutionStrategyProvider;
END_VAR
VAR
	graphInstance : I_GraphInstance;
END_VAR
DisposeGraphInstance(InstanceId);
graphInstance := CreateNewGraphInstance(InstanceId, Graph, InstanceExecutionStrategyProvider);
graphInstances.AddOrUpdate(InstanceId, graphInstance);
EmitOnGraphInstanceAddedEvent(graphInstance);
AddNewGraphInstance := graphInstance;
END_METHOD

METHOD PUBLIC CyclicCall
VAR
	graphInstance : I_GraphInstance;
END_VAR
IF NOT enumerator.IsValid THEN
	GetNewEnumerator();
ELSE
	enumerator.Reset();
END_IF

WHILE (enumerator.MoveNext()) DO
	
	IF enumerator.TryGet(graphInstance) THEN
		graphInstance.CyclicCall();
	END_IF

END_WHILE
END_METHOD

METHOD PUBLIC DisposeAll
VAR
	graphInstance : I_GraphInstance;
END_VAR
IF NOT enumerator.IsValid THEN
	GetNewEnumerator();
ELSE
	enumerator.Reset();
END_IF

WHILE enumerator.MoveNext() DO
	IF enumerator.TryGet(graphInstance) THEN
		graphInstance.Dispose();
	END_IF
END_WHILE

graphInstances.Clear();
END_METHOD

METHOD PUBLIC DisposeDefaultGraphInstance
DisposeGraphInstance(DEFAULT_ID);
END_METHOD

METHOD PUBLIC DisposeGraphInstance
VAR_INPUT
	InstanceId : T_MAXSTRING;
END_VAR
VAR
	graphInstance : I_GraphInstance;
END_VAR
IF NOT graphInstances.TryGetValue(InstanceId, graphInstance) THEN
	RETURN;
END_IF

graphInstances.Remove(InstanceId);

IF graphInstance = 0 THEN
	RETURN;
END_IF

graphInstance.Dispose();
END_METHOD

METHOD PUBLIC SerializeWith
VAR_INPUT
	Serializer : I_Serializer;
END_VAR
VAR
	graphInstance : I_GraphInstance;
END_VAR
IF graphInstances.IsEmpty THEN
	RETURN;
END_IF

Serializer.AddKey('graphInstances');
Serializer.StartArray();

IF NOT enumerator.IsValid THEN
	GetNewEnumerator();
ELSE
	enumerator.Reset();
END_IF

WHILE enumerator.MoveNext() DO
	IF enumerator.TryGet(graphInstance) THEN
		graphInstance.SerializeWith(Serializer);
	END_IF
END_WHILE

Serializer.EndArray();
END_METHOD

METHOD PUBLIC TryGetDefaultGraphInstance : BOOL
VAR_INPUT
	Destination : REFERENCE TO I_GraphInstance;
END_VAR
TryGetDefaultGraphInstance := TryGetGraphInstance(DEFAULT_ID, Destination);
END_METHOD

METHOD PUBLIC TryGetGraphInstance : BOOL
VAR_INPUT
	InstanceId : T_MAXSTRING;
	Destination : REFERENCE TO I_GraphInstance;
END_VAR
VAR
	graphInstance : I_GraphInstance;
END_VAR
IF NOT graphInstances.TryGetValue(InstanceId, graphInstance) THEN
	RETURN;
END_IF

Destination := graphInstance;
TryGetGraphInstance := TRUE;
END_METHOD

END_FUNCTION_BLOCK

// GraphInstance/GraphInstance/GraphInstance
{attribute 'linkalways'} 
{attribute 'no_explicit_call' := 'This FB is a CLASS and must be accessed using methods or properties'}
{attribute 'enable_dynamic_creation'}
FUNCTION_BLOCK GraphInstance EXTENDS Disposable IMPLEMENTS I_GraphInstance
VAR
	_id : T_MAXSTRING;
	_graph : I_Graph;
	executionStrategy : I_GraphExecutionStrategy;
END_VAR

METHOD FB_init : BOOL
VAR_INPUT
	bInitRetains : BOOL; // if TRUE, the retain variables are initialized (warm start / cold start)
	bInCopyCode : BOOL;  // if TRUE, the instance afterwards gets moved into the copy code (online change)
	Id : T_MAXSTRING;
	TargetGraph : I_Graph;
	ExecutionStrategyProvider : I_GraphExecutionStrategyProvider;
END_VAR
THIS^._id := Id;
THIS^._graph := TargetGraph;
THIS^.executionStrategy := ExecutionStrategyProvider.Create(TargetGraph);
END_METHOD

METHOD FB_exit : BOOL
VAR_INPUT
	bInCopyCode : BOOL; // if TRUE, the exit method is called for exiting an instance that is copied afterwards (online change).
END_VAR
IF bInCopyCode THEN
	RETURN;
END_IF

IF executionStrategy <> 0 THEN
	executionStrategy.Dispose();
	executionStrategy := 0;
END_IF

IF _graph <> 0 THEN
	_graph.Dispose();
	_graph := 0;
END_IF
END_METHOD

METHOD PUBLIC Accept
VAR_INPUT
	Visitor : I_GraphInstanceVisitor;
END_VAR
Visitor.VisitGraphInstance(THIS^);
END_METHOD

PROPERTY PUBLIC CycleCount : UDINT
GET
CycleCount := executionStrategy.CycleCount;
END_GET
END_PROPERTY

METHOD PUBLIC CyclicCall
VAR_INPUT
END_VAR
executionStrategy.CyclicCall();
END_METHOD

PROPERTY PUBLIC Graph : I_Graph
GET
Graph := _graph;
END_GET
END_PROPERTY

PROPERTY PUBLIC Id : T_MAXSTRING
GET
Id := _id;
END_GET
END_PROPERTY

PROPERTY PUBLIC IsEndOfCycle : BOOL
GET
IsEndOfCycle := executionStrategy.IsEndOfCycle;
END_GET
END_PROPERTY

PROPERTY PUBLIC IsRunning : BOOL
GET
IsRunning := executionStrategy.IsRunning;
END_GET
END_PROPERTY

PROPERTY PUBLIC IsStopped : BOOL
GET
IsStopped := executionStrategy.IsStopped;
END_GET
END_PROPERTY

METHOD PUBLIC SerializeWith
VAR_INPUT
	Serializer : I_Serializer;
END_VAR
VAR
	graphInstance : I_GraphInstance;
END_VAR
Serializer.StartObject();
Serializer.AddKeyString('id', _id);
Serializer.AddKeyObject('graph', _graph);
Serializer.EndObject();
END_METHOD

METHOD Start
VAR_INPUT
END_VAR
executionStrategy.Start();
END_METHOD

METHOD Stop
VAR_INPUT
END_VAR
executionStrategy.Stop();
END_METHOD

END_FUNCTION_BLOCK

// GraphInstance/Events/GraphInstanceAddedEvent
{attribute 'linkalways'} 
{attribute 'no_explicit_call' := 'This FB is a CLASS and must be accessed using methods or properties'}
{attribute 'enable_dynamic_creation'}
FUNCTION_BLOCK GraphInstanceAddedEvent EXTENDS Disposable IMPLEMENTS I_GraphInstanceAddedEvent
VAR
	_target : I_GraphInstance;
END_VAR

METHOD FB_init : BOOL
VAR_INPUT
	bInitRetains : BOOL; // if TRUE, the retain variables are initialized (warm start / cold start)
	bInCopyCode : BOOL;  // if TRUE, the instance afterwards gets moved into the copy code (online change)
	Target : I_GraphInstance;
END_VAR
THIS^._target := Target;
END_METHOD

PROPERTY PUBLIC Target : I_GraphInstance
GET
Target := _target;
END_GET
END_PROPERTY

END_FUNCTION_BLOCK

// GraphInstance/Events/I_GraphInstanceAddedEvent
INTERFACE I_GraphInstanceAddedEvent EXTENDS I_Event

PROPERTY PUBLIC Target : I_GraphInstance
GET
END_GET
END_PROPERTY

END_INTERFACE

// API/Visitors/GetStatusVisitor
{attribute 'linkalways'} 
{attribute 'no_explicit_call' := 'This FB is a CLASS and must be accessed using methods or properties'}
{attribute 'enable_dynamic_creation'}
FUNCTION_BLOCK GetStatusVisitor IMPLEMENTS I_GraphVisitor, I_NodeVisitor, I_ExtensionVisitor, I_ContentVisitor, I_AlarmVisitor
VAR
	serializer : I_Serializer;
END_VAR

METHOD PUBLIC Initialize
VAR_INPUT
	Serializer : I_Serializer;
END_VAR
THIS^.serializer := Serializer;
END_METHOD

METHOD VisitAlarm
VAR_INPUT
	VisitingAlarm : I_Alarm;
END_VAR
IF VisitingAlarm.Active THEN
	serializer.StartObject();
	serializer.AddKeyString('message', VisitingAlarm.Message);
	serializer.AddKeyString('reason', VisitingAlarm.Reason);
	serializer.EndObject();
END_IF
END_METHOD

METHOD VisitContent
VAR_INPUT
	VisitingContent : I_Content;
END_VAR
serializer.StartObject();

serializer.AddKeyString('name', VisitingContent.Name);
serializer.AddKeyObject('value', VisitingContent.Data);

serializer.EndObject();
END_METHOD

METHOD VisitExtension
VAR_INPUT
	VisitingExtension : I_Extension;
END_VAR
Serializer.StartObject();
Serializer.AddKeyString('name', VisitingExtension.Name);

IF VisitingExtension.Alarms.HasAlarms THEN
	serializer.addkey('alarms');
	serializer.StartArray();
	VisitingExtension.Alarms.Accept(THIS^);
	serializer.EndArray();
END_IF

IF VisitingExtension.Contents.HasContents THEN
	serializer.addkey('contents');
	serializer.StartArray();
	VisitingExtension.Contents.Accept(THIS^);
	serializer.EndArray();
END_IF

Serializer.EndObject();
END_METHOD

METHOD VisitGraph
VAR_INPUT
	VisitingGraph : I_Graph;
END_VAR
VAR
	includeInGetStatusVisitor : IncludeInGetStatusVisitor;
END_VAR
serializer.StartObject();

serializer.addKeyString('uuid', VisitingGraph.Uuid);

IF VisitingGraph.Alarms.HasRaisedAlarm THEN
	serializer.addkey('alarms');
	serializer.StartArray();
	VisitingGraph.Alarms.Accept(THIS^);
	serializer.EndArray();
END_IF

IF includeInGetStatusVisitor.CheckExtensions(VisitingGraph) THEN
	serializer.addkey('extensions');
	serializer.StartArray();
	VisitingGraph.Extensions.Accept(THIS^);
	serializer.EndArray();
END_IF

IF VisitingGraph.Contents.HasContents THEN
	serializer.addkey('contents');
	serializer.StartArray();
	VisitingGraph.Contents.Accept(THIS^);
	serializer.EndArray();
END_IF

IF VisitingGraph.Nodes.HasNodes THEN
	serializer.addkey('nodes');
	serializer.StartArray();
	VisitingGraph.Nodes.Accept(THIS^);
	serializer.EndArray();
END_IF

serializer.EndObject();
END_METHOD

METHOD VisitNode
VAR_INPUT
	VisitingNode : I_Node;
END_VAR
VAR
	includeInGetStatusVisitor : IncludeInGetStatusVisitor;
END_VAR
IF NOT includeInGetStatusVisitor.CheckNode(VisitingNode) THEN
	RETURN;
END_IF

serializer.StartObject();
serializer.addKeyString('id', VisitingNode.Id);

IF VisitingNode.Alarms.HasRaisedAlarm THEN
	serializer.addkey('alarms');
	serializer.StartArray();
	VisitingNode.Alarms.Accept(THIS^);
	serializer.EndArray();
END_IF

IF includeInGetStatusVisitor.CheckExtensions(VisitingNode) THEN
	serializer.addkey('extensions');
	serializer.StartArray();
	VisitingNode.Extensions.Accept(THIS^);
	serializer.EndArray();
END_IF

IF VisitingNode.Contents.HasContents THEN
	serializer.addkey('contents');
	serializer.StartArray();
	VisitingNode.Contents.Accept(THIS^);
	serializer.EndArray();
END_IF

serializer.EndObject();
END_METHOD

END_FUNCTION_BLOCK

// API/Visitors/IncludeInGetStatusVisitor
{attribute 'linkalways'} 
{attribute 'no_explicit_call' := 'This FB is a CLASS and must be accessed using methods or properties'}
{attribute 'enable_dynamic_creation'}
FUNCTION_BLOCK IncludeInGetStatusVisitor IMPLEMENTS I_NodeVisitor, I_ExtensionVisitor
VAR
	shouldInclude : BOOL;
END_VAR

METHOD PUBLIC CheckExtensions : BOOL;
VAR_INPUT
	ExtensionHost : I_HostExtensions;
END_VAR
shouldInclude := FALSE;
ExtensionHost.Extensions.Accept(THIS^);
CheckExtensions := shouldInclude;
END_METHOD

METHOD PUBLIC CheckNode : BOOL;
VAR_INPUT
	Node : I_Node;
END_VAR
shouldInclude := FALSE;
Node.Accept(THIS^);
CheckNode := shouldInclude;
END_METHOD

METHOD VisitExtension
VAR_INPUT
	VisitingExtension : I_Extension;
END_VAR
IF VisitingExtension.Contents.HasContents THEN
	shouldInclude := TRUE;
	RETURN;
END_IF

IF VisitingExtension.Alarms.HasRaisedAlarm THEN
	shouldInclude := TRUE;
	RETURN;
END_IF
END_METHOD

METHOD VisitNode
VAR_INPUT
	VisitingNode : I_Node;
END_VAR
IF VisitingNode.Contents.HasContents THEN
	shouldInclude := TRUE;
	RETURN;
END_IF

IF VisitingNode.Alarms.HasRaisedAlarm THEN
	shouldInclude := TRUE;
	RETURN;
END_IF

IF VisitingNode.Extensions.HasExtensions THEN
	VisitingNode.Extensions.Accept(THIS^);
END_IF
END_METHOD

END_FUNCTION_BLOCK

// API/Handlers/GetBlueprintsRpcHandler
{attribute 'linkalways'} 
{attribute 'no_explicit_call' := 'This FB is a CLASS and must be accessed using methods or properties'}
{attribute 'enable_dynamic_creation'}
FUNCTION_BLOCK GetBlueprintsRpcHandler IMPLEMENTS I_AsynchronousRpcHandler
VAR
	graphFramework : I_GraphFramework;
END_VAR

METHOD Handle
VAR_INPUT
	Parameters : I_Deserializer;
	Response : I_AsynchronousRpcResponse;
END_VAR
VAR
	getBlueprintsVisitor : GetBlueprintsVisitor;
	getPaginatedBlueprintsVisitor : GetPaginatedBlueprintsVisitor;
	visitor : I_NodeFactoryVisitor;
	serializer : I_Serializer;
	feedback : DeserializerFeedback;
	offset : UDINT;
	maxLimit : UDINT;
END_VAR
IF graphFramework = 0 THEN
	Response.RejectWithError('INTERNAL_ERROR','GetBlueprintsRpcHandler has not been correctly initialized');
	RETURN;
END_IF

serializer := Response.GetSerializer();

IF Parameters.TryGetKeyUdint('offset', offset, feedback) AND_THEN Parameters.TryGetKeyUdint('limit', maxLimit, feedback) THEN
	// if the offset and limit are provide then use the paginated visitor
	getPaginatedBlueprintsVisitor.Initialize(serializer, offset, maxlimit);
	visitor := getPaginatedBlueprintsVisitor;
ELSE
	// if the offset and limit are not supplied then try to get all blueprints
	getBlueprintsVisitor.Initialize(serializer);
	visitor := getBlueprintsVisitor;
END_IF

graphFramework.NodeFactory.Accept(visitor);
Response.CompleteWithSerializer(serializer);
serializer.Dispose();
END_METHOD

METHOD PUBLIC Initialize
VAR_INPUT
	GraphFramework : I_GraphFramework;
END_VAR
THIS^.graphFramework := GraphFramework;
END_METHOD

END_FUNCTION_BLOCK

// API/Visitors/GetPaginatedBlueprintsVisitor
{attribute 'linkalways'} 
{attribute 'no_explicit_call' := 'This FB is a CLASS and must be accessed using methods or properties'}
{attribute 'enable_dynamic_creation'}
FUNCTION_BLOCK GetPaginatedBlueprintsVisitor IMPLEMENTS I_NodeFactoryVisitor, I_NodePrototypeVisitor, I_NodeVisitor, I_ExtensionVisitor, I_InputPortVisitor, I_OutputPortVisitor, I_MetadataVisitor, I_ContentVisitor, I_ParameterVisitor, I_AlarmVisitor
VAR
	serializer : I_Serializer;
	offset : UDINT;
	maxLimit : UDINT;
	
	// used to track count
	currentIndex : UDINT;
	endIndex : UDINT;
	blueprintsCollected : UDINT;
	totalBlueprints : UDINT;
END_VAR

METHOD PUBLIC Initialize
VAR_INPUT
	Serializer : I_Serializer;
	Offset : UDINT;
	MaxLimit : UDINT;
END_VAR
THIS^.serializer := Serializer;
THIS^.offset := Offset;
THIS^.maxLimit := MaxLimit;

THIS^.currentIndex := 0;
THIS^.endIndex := Offset + MaxLimit -1;

THIS^.blueprintsCollected := 0;
THIS^.totalBlueprints := 0;
END_METHOD

METHOD VisitAlarm
VAR_INPUT
	VisitingAlarm : I_Alarm;
END_VAR
serializer.AddString(VisitingAlarm.Message);
END_METHOD

METHOD VisitContent
VAR_INPUT
	VisitingContent : I_Content;
END_VAR
serializer.StartObject();

serializer.AddKeyString('name', VisitingContent.Name);
serializer.Addkey('datatype');
VisitingContent.Data.SerializeTypeWith(serializer);

IF VisitingContent.Metadatum.HasMetadata THEN
	serializer.addkey('metadata');
	serializer.StartArray();
	VisitingContent.Metadatum.Accept(THIS^);
	serializer.EndArray();
END_IF

serializer.EndObject();
END_METHOD

METHOD VisitExtension
VAR_INPUT
	VisitingExtension : I_Extension;
END_VAR
Serializer.StartObject();
Serializer.AddKeyString('name', VisitingExtension.Name);

IF VisitingExtension.Metadatum.HasMetadata THEN
	serializer.addkey('metadata');
	serializer.StartArray();
	VisitingExtension.Metadatum.Accept(THIS^);
	serializer.EndArray();
END_IF

